    movel([0.121512, -1.277882, -2.639654, -0.794853, 1.570796, 1.692308],accel_mss,speed_ms,0,blend_radius_m)
    movel([0.121915, -1.277664, -2.639778, -0.794948, 1.570796, 1.692711],accel_mss,speed_ms,0,blend_radius_m)
    movel([0.122224, -1.277485, -2.639879, -0.795025, 1.570796, 1.693020],accel_mss,speed_ms,0,blend_radius_m)
    movel([0.122594, -1.277272, -2.639999, -0.795118, 1.570796, 1.693390],accel_mss,speed_ms,0,blend_radius_m)
    movel([0.122927, -1.277174, -2.640055, -0.795160, 1.570796, 1.693724],accel_mss,speed_ms,0,blend_radius_m)
    movel([0.123154, -1.277358, -2.639950, -0.795080, 1.570796, 1.693950],accel_mss,speed_ms,0,blend_radius_m)
    movel([0.122937, -1.277676, -2.639771, -0.794942, 1.570796, 1.693733],accel_mss,speed_ms,0,blend_radius_m)
    movel([0.122394, -1.277926, -2.639629, -0.794834, 1.570796, 1.693190],accel_mss,speed_ms,0,blend_radius_m)
    movel([0.122493, -1.278132, -2.639513, -0.794745, 1.570796, 1.693289],accel_mss,speed_ms,0,blend_radius_m)
    movel([0.122823, -1.278090, -2.639536, -0.794763, 1.570796, 1.693620],accel_mss,speed_ms,0,blend_radius_m)
    movel([0.123129, -1.277991, -2.639592, -0.794806, 1.570796, 1.693926],accel_mss,speed_ms,0,blend_radius_m)
    movel([0.123433, -1.277648, -2.639786, -0.794954, 1.570796, 1.694230],accel_mss,speed_ms,0,blend_radius_m)
    movel([0.123760, -1.277440, -2.639904, -0.795045, 1.570796, 1.694556],accel_mss,speed_ms,0,blend_radius_m)
    movel([0.124094, -1.277452, -2.639898, -0.795040, 1.570796, 1.694890],accel_mss,speed_ms,0,blend_radius_m)
    movel([0.124564, -1.277440, -2.639904, -0.795045, 1.570796, 1.695360],accel_mss,speed_ms,0,blend_radius_m)
    movel([0.125059, -1.277384, -2.639936, -0.795069, 1.570796, 1.695855],accel_mss,speed_ms,0,blend_radius_m)
    movel([0.125372, -1.277273, -2.639999, -0.795117, 1.570796, 1.696168],accel_mss,speed_ms,0,blend_radius_m)
    movel([0.125657, -1.277244, -2.640015, -0.795130, 1.570796, 1.696454],accel_mss,speed_ms,0,blend_radius_m)
    movel([0.125972, -1.277065, -2.640117, -0.795208, 1.570796, 1.696768],accel_mss,speed_ms,0,blend_radius_m)
    movel([0.126196, -1.277124, -2.640083, -0.795182, 1.570796, 1.696993],accel_mss,speed_ms,0,blend_radius_m)
    movel([0.126436, -1.277173, -2.640055, -0.795161, 1.570796, 1.697232],accel_mss,speed_ms,0,blend_radius_m)
    movel([0.126810, -1.277070, -2.640113, -0.795205, 1.570796, 1.697606],accel_mss,speed_ms,0,blend_radius_m)
    movel([0.127277, -1.276889, -2.640215, -0.795284, 1.570796, 1.698073],accel_mss,speed_ms,0,blend_radius_m)
    movel([0.127645, -1.276791, -2.640271, -0.795327, 1.570796, 1.698441],accel_mss,speed_ms,0,blend_radius_m)
    movel([0.128058, -1.276835, -2.640246, -0.795308, 1.570796, 1.698854],accel_mss,speed_ms,0,blend_radius_m)
    movel([0.128268, -1.276992, -2.640157, -0.795239, 1.570796, 1.699064],accel_mss,speed_ms,0,blend_radius_m)
    movel([0.128442, -1.277211, -2.640033, -0.795144, 1.570796, 1.699239],accel_mss,speed_ms,0,blend_radius_m)
    movel([0.128502, -1.277437, -2.639906, -0.795046, 1.570796, 1.699298],accel_mss,speed_ms,0,blend_radius_m)
    movel([0.128278, -1.277739, -2.639735, -0.794915, 1.570796, 1.699074],accel_mss,speed_ms,0,blend_radius_m)
    movel([0.128301, -1.278030, -2.639570, -0.794789, 1.570796, 1.699097],accel_mss,speed_ms,0,blend_radius_m)
    movel([0.128456, -1.278253, -2.639444, -0.794692, 1.570796, 1.699252],accel_mss,speed_ms,0,blend_radius_m)
    movel([0.128142, -1.278841, -2.639111, -0.794438, 1.570796, 1.698939],accel_mss,speed_ms,0,blend_radius_m)
    movel([0.127643, -1.279450, -2.638765, -0.794174, 1.570796, 1.698439],accel_mss,speed_ms,0,blend_radius_m)
    movel([0.127331, -1.279820, -2.638555, -0.794015, 1.570796, 1.698128],accel_mss,speed_ms,0,blend_radius_m)
    movel([0.127066, -1.280148, -2.638368, -0.793873, 1.570796, 1.697863],accel_mss,speed_ms,0,blend_radius_m)
    movel([0.126852, -1.280424, -2.638211, -0.793754, 1.570796, 1.697648],accel_mss,speed_ms,0,blend_radius_m)
    movel([0.126937, -1.280641, -2.638087, -0.793661, 1.570796, 1.697734],accel_mss,speed_ms,0,blend_radius_m)
    movel([0.127240, -1.280865, -2.637959, -0.793565, 1.570796, 1.698036],accel_mss,speed_ms,0,blend_radius_m)
    movel([0.127528, -1.281108, -2.637821, -0.793460, 1.570796, 1.698325],accel_mss,speed_ms,0,blend_radius_m)
    movel([0.127643, -1.281364, -2.637675, -0.793350, 1.570796, 1.698439],accel_mss,speed_ms,0,blend_radius_m)
    movel([0.127335, -1.281559, -2.637563, -0.793266, 1.570796, 1.698131],accel_mss,speed_ms,0,blend_radius_m)
    movel([0.127124, -1.281455, -2.637623, -0.793311, 1.570796, 1.697920],accel_mss,speed_ms,0,blend_radius_m)
    movel([0.126991, -1.281268, -2.637730, -0.793391, 1.570796, 1.697788],accel_mss,speed_ms,0,blend_radius_m)
    movel([0.126865, -1.281079, -2.637837, -0.793473, 1.570796, 1.697661],accel_mss,speed_ms,0,blend_radius_m)
    movel([0.126558, -1.281192, -2.637773, -0.793424, 1.570796, 1.697354],accel_mss,speed_ms,0,blend_radius_m)
    movel([0.126435, -1.280994, -2.637886, -0.793509, 1.570796, 1.697231],accel_mss,speed_ms,0,blend_radius_m)
    movel([0.126185, -1.280895, -2.637942, -0.793552, 1.570796, 1.696981],accel_mss,speed_ms,0,blend_radius_m)
    movel([0.126273, -1.280615, -2.638102, -0.793672, 1.570796, 1.697069],accel_mss,speed_ms,0,blend_radius_m)
    movel([0.126374, -1.280318, -2.638271, -0.793800, 1.570796, 1.697170],accel_mss,speed_ms,0,blend_radius_m)
    movel([0.126672, -1.280154, -2.638364, -0.793870, 1.570796, 1.697468],accel_mss,speed_ms,0,blend_radius_m)
    movel([0.126485, -1.280006, -2.638449, -0.793935, 1.570796, 1.697281],accel_mss,speed_ms,0,blend_radius_m)
    movel([0.126217, -1.280245, -2.638312, -0.793831, 1.570796, 1.697013],accel_mss,speed_ms,0,blend_radius_m)
    movel([0.125927, -1.280465, -2.638187, -0.793737, 1.570796, 1.696723],accel_mss,speed_ms,0,blend_radius_m)
    movel([0.125642, -1.280712, -2.638046, -0.793630, 1.570796, 1.696438],accel_mss,speed_ms,0,blend_radius_m)
    movel([0.125248, -1.280906, -2.637936, -0.793547, 1.570796, 1.696044],accel_mss,speed_ms,0,blend_radius_m)
    movel([0.124945, -1.281110, -2.637820, -0.793459, 1.570796, 1.695741],accel_mss,speed_ms,0,blend_radius_m)
    movel([0.124618, -1.281268, -2.637729, -0.793391, 1.570796, 1.695414],accel_mss,speed_ms,0,blend_radius_m)
    movel([0.124820, -1.281407, -2.637650, -0.793332, 1.570796, 1.695616],accel_mss,speed_ms,0,blend_radius_m)
    movel([0.125120, -1.281303, -2.637710, -0.793376, 1.570796, 1.695916],accel_mss,speed_ms,0,blend_radius_m)
    movel([0.125422, -1.281303, -2.637709, -0.793376, 1.570796, 1.696218],accel_mss,speed_ms,0,blend_radius_m)
    movel([0.125734, -1.281325, -2.637697, -0.793367, 1.570796, 1.696530],accel_mss,speed_ms,0,blend_radius_m)
    movel([0.125551, -1.281207, -2.637764, -0.793418, 1.570796, 1.696347],accel_mss,speed_ms,0,blend_radius_m)
    movel([0.125887, -1.281100, -2.637826, -0.793464, 1.570796, 1.696683],accel_mss,speed_ms,0,blend_radius_m)
    movel([0.126035, -1.281250, -2.637740, -0.793399, 1.570796, 1.696831],accel_mss,speed_ms,0,blend_radius_m)
    movel([0.126335, -1.281283, -2.637721, -0.793385, 1.570796, 1.697131],accel_mss,speed_ms,0,blend_radius_m)
    movel([0.126542, -1.281456, -2.637622, -0.793310, 1.570796, 1.697338],accel_mss,speed_ms,0,blend_radius_m)
    movel([0.126874, -1.281511, -2.637591, -0.793287, 1.570796, 1.697670],accel_mss,speed_ms,0,blend_radius_m)
    movel([0.127085, -1.281732, -2.637465, -0.793192, 1.570796, 1.697881],accel_mss,speed_ms,0,blend_radius_m)
    movel([0.126908, -1.282027, -2.637296, -0.793066, 1.570796, 1.697705],accel_mss,speed_ms,0,blend_radius_m)
    movel([0.126872, -1.282378, -2.637096, -0.792915, 1.570796, 1.697668],accel_mss,speed_ms,0,blend_radius_m)
    movel([0.126732, -1.282647, -2.636942, -0.792800, 1.570796, 1.697528],accel_mss,speed_ms,0,blend_radius_m)
    movel([0.127032, -1.282483, -2.637035, -0.792870, 1.570796, 1.697828],accel_mss,speed_ms,0,blend_radius_m)
    movel([0.127020, -1.282092, -2.637259, -0.793038, 1.570796, 1.697816],accel_mss,speed_ms,0,blend_radius_m)
    movel([0.127207, -1.281796, -2.637428, -0.793165, 1.570796, 1.698004],accel_mss,speed_ms,0,blend_radius_m)
    movel([0.127325, -1.281990, -2.637318, -0.793082, 1.570796, 1.698121],accel_mss,speed_ms,0,blend_radius_m)
    movel([0.127108, -1.282326, -2.637125, -0.792937, 1.570796, 1.697904],accel_mss,speed_ms,0,blend_radius_m)
    movel([0.127401, -1.282233, -2.637178, -0.792977, 1.570796, 1.698197],accel_mss,speed_ms,0,blend_radius_m)
    movel([0.127190, -1.282793, -2.636858, -0.792738, 1.570796, 1.697986],accel_mss,speed_ms,0,blend_radius_m)
    movel([0.126973, -1.283052, -2.636710, -0.792627, 1.570796, 1.697769],accel_mss,speed_ms,0,blend_radius_m)
    movel([0.126665, -1.283232, -2.636607, -0.792550, 1.570796, 1.697462],accel_mss,speed_ms,0,blend_radius_m)
    movel([0.126509, -1.283540, -2.636430, -0.792419, 1.570796, 1.697305],accel_mss,speed_ms,0,blend_radius_m)
    movel([0.126164, -1.283969, -2.636184, -0.792236, 1.570796, 1.696960],accel_mss,speed_ms,0,blend_radius_m)
    movel([0.125846, -1.284341, -2.635970, -0.792077, 1.570796, 1.696642],accel_mss,speed_ms,0,blend_radius_m)
    movel([0.126192, -1.284417, -2.635927, -0.792045, 1.570796, 1.696988],accel_mss,speed_ms,0,blend_radius_m)
    movel([0.126470, -1.284556, -2.635847, -0.791986, 1.570796, 1.697267],accel_mss,speed_ms,0,blend_radius_m)
    movel([0.126536, -1.284775, -2.635721, -0.791893, 1.570796, 1.697332],accel_mss,speed_ms,0,blend_radius_m)
    movel([0.126661, -1.284987, -2.635599, -0.791803, 1.570796, 1.697458],accel_mss,speed_ms,0,blend_radius_m)
    movel([0.126532, -1.285317, -2.635409, -0.791663, 1.570796, 1.697328],accel_mss,speed_ms,0,blend_radius_m)
    movel([0.126278, -1.285671, -2.635205, -0.791513, 1.570796, 1.697074],accel_mss,speed_ms,0,blend_radius_m)
    movel([0.125958, -1.286079, -2.634970, -0.791340, 1.570796, 1.696754],accel_mss,speed_ms,0,blend_radius_m)
    movel([0.125587, -1.286339, -2.634821, -0.791230, 1.570796, 1.696383],accel_mss,speed_ms,0,blend_radius_m)
    movel([0.125858, -1.286124, -2.634944, -0.791320, 1.570796, 1.696654],accel_mss,speed_ms,0,blend_radius_m)
    movel([0.125869, -1.285839, -2.635109, -0.791441, 1.570796, 1.696665],accel_mss,speed_ms,0,blend_radius_m)
    movel([0.126028, -1.285541, -2.635280, -0.791568, 1.570796, 1.696825],accel_mss,speed_ms,0,blend_radius_m)
    movel([0.126232, -1.285026, -2.635577, -0.791786, 1.570796, 1.697029],accel_mss,speed_ms,0,blend_radius_m)
    movel([0.126003, -1.284962, -2.635614, -0.791813, 1.570796, 1.696799],accel_mss,speed_ms,0,blend_radius_m)
    movel([0.125957, -1.284696, -2.635767, -0.791927, 1.570796, 1.696753],accel_mss,speed_ms,0,blend_radius_m)
    movel([0.125809, -1.284543, -2.635854, -0.791991, 1.570796, 1.696605],accel_mss,speed_ms,0,blend_radius_m)
    movel([0.125586, -1.284429, -2.635920, -0.792040, 1.570796, 1.696383],accel_mss,speed_ms,0,blend_radius_m)
    movel([0.125377, -1.284351, -2.635965, -0.792073, 1.570796, 1.696173],accel_mss,speed_ms,0,blend_radius_m)
    movel([0.125610, -1.284068, -2.636127, -0.792194, 1.570796, 1.696406],accel_mss,speed_ms,0,blend_radius_m)
    movel([0.125992, -1.283659, -2.636362, -0.792368, 1.570796, 1.696789],accel_mss,speed_ms,0,blend_radius_m)
    movel([0.126321, -1.283308, -2.636563, -0.792518, 1.570796, 1.697118],accel_mss,speed_ms,0,blend_radius_m)
    movel([0.126533, -1.282968, -2.636758, -0.792663, 1.570796, 1.697330],accel_mss,speed_ms,0,blend_radius_m)
    movel([0.126193, -1.283188, -2.636632, -0.792569, 1.570796, 1.696989],accel_mss,speed_ms,0,blend_radius_m)
    movel([0.125766, -1.283548, -2.636426, -0.792415, 1.570796, 1.696563],accel_mss,speed_ms,0,blend_radius_m)
    movel([0.125446, -1.283919, -2.636213, -0.792257, 1.570796, 1.696242],accel_mss,speed_ms,0,blend_radius_m)
    movel([0.125139, -1.284055, -2.636135, -0.792199, 1.570796, 1.695935],accel_mss,speed_ms,0,blend_radius_m)
    movel([0.124558, -1.284490, -2.635885, -0.792014, 1.570796, 1.695354],accel_mss,speed_ms,0,blend_radius_m)
    movel([0.124536, -1.284797, -2.635709, -0.791884, 1.570796, 1.695333],accel_mss,speed_ms,0,blend_radius_m)
    movel([0.124872, -1.284837, -2.635685, -0.791866, 1.570796, 1.695668],accel_mss,speed_ms,0,blend_radius_m)
    movel([0.125134, -1.284821, -2.635695, -0.791873, 1.570796, 1.695931],accel_mss,speed_ms,0,blend_radius_m)
    movel([0.125420, -1.284693, -2.635768, -0.791928, 1.570796, 1.696217],accel_mss,speed_ms,0,blend_radius_m)
    movel([0.125608, -1.284848, -2.635679, -0.791862, 1.570796, 1.696404],accel_mss,speed_ms,0,blend_radius_m)
    movel([0.125786, -1.285070, -2.635551, -0.791768, 1.570796, 1.696583],accel_mss,speed_ms,0,blend_radius_m)
    movel([0.125996, -1.285162, -2.635498, -0.791728, 1.570796, 1.696792],accel_mss,speed_ms,0,blend_radius_m)
    movel([0.125747, -1.285560, -2.635269, -0.791559, 1.570796, 1.696543],accel_mss,speed_ms,0,blend_radius_m)
    movel([0.125404, -1.285997, -2.635017, -0.791374, 1.570796, 1.696200],accel_mss,speed_ms,0,blend_radius_m)
    movel([0.125296, -1.286269, -2.634861, -0.791259, 1.570796, 1.696093],accel_mss,speed_ms,0,blend_radius_m)
    movel([0.124953, -1.286578, -2.634682, -0.791128, 1.570796, 1.695749],accel_mss,speed_ms,0,blend_radius_m)
    movel([0.124458, -1.286900, -2.634496, -0.790992, 1.570796, 1.695255],accel_mss,speed_ms,0,blend_radius_m)
    movel([0.123806, -1.287353, -2.634235, -0.790801, 1.570796, 1.694603],accel_mss,speed_ms,0,blend_radius_m)
    movel([0.124318, -1.287180, -2.634335, -0.790874, 1.570796, 1.695114],accel_mss,speed_ms,0,blend_radius_m)
    movel([0.124661, -1.287037, -2.634417, -0.790935, 1.570796, 1.695458],accel_mss,speed_ms,0,blend_radius_m)
    movel([0.124937, -1.286829, -2.634537, -0.791022, 1.570796, 1.695733],accel_mss,speed_ms,0,blend_radius_m)
    movel([0.125165, -1.286556, -2.634695, -0.791138, 1.570796, 1.695962],accel_mss,speed_ms,0,blend_radius_m)
    movel([0.125011, -1.286951, -2.634467, -0.790971, 1.570796, 1.695807],accel_mss,speed_ms,0,blend_radius_m)
    movel([0.124648, -1.287248, -2.634295, -0.790845, 1.570796, 1.695444],accel_mss,speed_ms,0,blend_radius_m)
    movel([0.124301, -1.287457, -2.634174, -0.790757, 1.570796, 1.695097],accel_mss,speed_ms,0,blend_radius_m)
    movel([0.123990, -1.287729, -2.634017, -0.790643, 1.570796, 1.694786],accel_mss,speed_ms,0,blend_radius_m)
    movel([0.123623, -1.287713, -2.634026, -0.790649, 1.570796, 1.694419],accel_mss,speed_ms,0,blend_radius_m)
    movel([0.123370, -1.287684, -2.634043, -0.790662, 1.570796, 1.694166],accel_mss,speed_ms,0,blend_radius_m)
    movel([0.122926, -1.288007, -2.633857, -0.790526, 1.570796, 1.693723],accel_mss,speed_ms,0,blend_radius_m)
    movel([0.122673, -1.288254, -2.633713, -0.790422, 1.570796, 1.693469],accel_mss,speed_ms,0,blend_radius_m)
    movel([0.122307, -1.288149, -2.633774, -0.790466, 1.570796, 1.693104],accel_mss,speed_ms,0,blend_radius_m)
    movel([0.122004, -1.288212, -2.633738, -0.790440, 1.570796, 1.692801],accel_mss,speed_ms,0,blend_radius_m)
    movel([0.121661, -1.288494, -2.633574, -0.790321, 1.570796, 1.692457],accel_mss,speed_ms,0,blend_radius_m)
    movel([0.121351, -1.288684, -2.633464, -0.790241, 1.570796, 1.692148],accel_mss,speed_ms,0,blend_radius_m)
    movel([0.121025, -1.288902, -2.633338, -0.790150, 1.570796, 1.691821],accel_mss,speed_ms,0,blend_radius_m)
    movel([0.120795, -1.289136, -2.633201, -0.790051, 1.570796, 1.691591],accel_mss,speed_ms,0,blend_radius_m)
    movel([0.120927, -1.288831, -2.633379, -0.790179, 1.570796, 1.691724],accel_mss,speed_ms,0,blend_radius_m)
    movel([0.120541, -1.288762, -2.633419, -0.790208, 1.570796, 1.691337],accel_mss,speed_ms,0,blend_radius_m)
    movel([0.120155, -1.288905, -2.633336, -0.790148, 1.570796, 1.690951],accel_mss,speed_ms,0,blend_radius_m)
    movel([0.119775, -1.289045, -2.633255, -0.790089, 1.570796, 1.690571],accel_mss,speed_ms,0,blend_radius_m)
    movel([0.119308, -1.289155, -2.633191, -0.790043, 1.570796, 1.690104],accel_mss,speed_ms,0,blend_radius_m)
    movel([0.119086, -1.289030, -2.633263, -0.790096, 1.570796, 1.689882],accel_mss,speed_ms,0,blend_radius_m)
    movel([0.118778, -1.288930, -2.633321, -0.790138, 1.570796, 1.689574],accel_mss,speed_ms,0,blend_radius_m)
    movel([0.118635, -1.288762, -2.633419, -0.790208, 1.570796, 1.689431],accel_mss,speed_ms,0,blend_radius_m)
    movel([0.118460, -1.288562, -2.633535, -0.790292, 1.570796, 1.689257],accel_mss,speed_ms,0,blend_radius_m)
    movel([0.118223, -1.288514, -2.633562, -0.790312, 1.570796, 1.689019],accel_mss,speed_ms,0,blend_radius_m)
    movel([0.118344, -1.288851, -2.633367, -0.790171, 1.570796, 1.689141],accel_mss,speed_ms,0,blend_radius_m)
    movel([0.118538, -1.289082, -2.633233, -0.790074, 1.570796, 1.689335],accel_mss,speed_ms,0,blend_radius_m)
    movel([0.118550, -1.289354, -2.633075, -0.789960, 1.570796, 1.689347],accel_mss,speed_ms,0,blend_radius_m)
    movel([0.118849, -1.289162, -2.633186, -0.790040, 1.570796, 1.689645],accel_mss,speed_ms,0,blend_radius_m)
    movel([0.118996, -1.289366, -2.633068, -0.789955, 1.570796, 1.689792],accel_mss,speed_ms,0,blend_radius_m)
    movel([0.118698, -1.289531, -2.632972, -0.789886, 1.570796, 1.689495],accel_mss,speed_ms,0,blend_radius_m)
    movel([0.118450, -1.289508, -2.632986, -0.789895, 1.570796, 1.689246],accel_mss,speed_ms,0,blend_radius_m)
    movel([0.118230, -1.289407, -2.633044, -0.789938, 1.570796, 1.689027],accel_mss,speed_ms,0,blend_radius_m)
    movel([0.118043, -1.289226, -2.633149, -0.790013, 1.570796, 1.688839],accel_mss,speed_ms,0,blend_radius_m)
    movel([0.117955, -1.289021, -2.633268, -0.790099, 1.570796, 1.688751],accel_mss,speed_ms,0,blend_radius_m)
    movel([0.118003, -1.288720, -2.633443, -0.790226, 1.570796, 1.688799],accel_mss,speed_ms,0,blend_radius_m)
    movel([0.118007, -1.288440, -2.633605, -0.790343, 1.570796, 1.688804],accel_mss,speed_ms,0,blend_radius_m)
    movel([0.118087, -1.288046, -2.633834, -0.790509, 1.570796, 1.688883],accel_mss,speed_ms,0,blend_radius_m)
    movel([0.118058, -1.287732, -2.634015, -0.790641, 1.570796, 1.688855],accel_mss,speed_ms,0,blend_radius_m)
    movel([0.117873, -1.287509, -2.634144, -0.790735, 1.570796, 1.688669],accel_mss,speed_ms,0,blend_radius_m)
    movel([0.117791, -1.287302, -2.634264, -0.790823, 1.570796, 1.688587],accel_mss,speed_ms,0,blend_radius_m)
    movel([0.117513, -1.287599, -2.634092, -0.790697, 1.570796, 1.688309],accel_mss,speed_ms,0,blend_radius_m)
    movel([0.117263, -1.287555, -2.634118, -0.790716, 1.570796, 1.688060],accel_mss,speed_ms,0,blend_radius_m)
    movel([0.116775, -1.287477, -2.634163, -0.790749, 1.570796, 1.687571],accel_mss,speed_ms,0,blend_radius_m)
    movel([0.116521, -1.287240, -2.634300, -0.790849, 1.570796, 1.687318],accel_mss,speed_ms,0,blend_radius_m)
    movel([0.116399, -1.286963, -2.634460, -0.790966, 1.570796, 1.687195],accel_mss,speed_ms,0,blend_radius_m)
    movel([0.116380, -1.286678, -2.634625, -0.791086, 1.570796, 1.687176],accel_mss,speed_ms,0,blend_radius_m)
    movel([0.116535, -1.286390, -2.634791, -0.791208, 1.570796, 1.687332],accel_mss,speed_ms,0,blend_radius_m)
    movel([0.116603, -1.286612, -2.634663, -0.791114, 1.570796, 1.687400],accel_mss,speed_ms,0,blend_radius_m)
    movel([0.116900, -1.286376, -2.634799, -0.791214, 1.570796, 1.687696],accel_mss,speed_ms,0,blend_radius_m)
    movel([0.116924, -1.286108, -2.634954, -0.791327, 1.570796, 1.687721],accel_mss,speed_ms,0,blend_radius_m)
    movel([0.116662, -1.286018, -2.635006, -0.791366, 1.570796, 1.687458],accel_mss,speed_ms,0,blend_radius_m)
    movel([0.117083, -1.285824, -2.635117, -0.791448, 1.570796, 1.687879],accel_mss,speed_ms,0,blend_radius_m)
    movel([0.117398, -1.285712, -2.635182, -0.791495, 1.570796, 1.688195],accel_mss,speed_ms,0,blend_radius_m)
    movel([0.117220, -1.285518, -2.635294, -0.791578, 1.570796, 1.688016],accel_mss,speed_ms,0,blend_radius_m)
    movel([0.116901, -1.285694, -2.635192, -0.791503, 1.570796, 1.687697],accel_mss,speed_ms,0,blend_radius_m)
    movel([0.117066, -1.285357, -2.635386, -0.791646, 1.570796, 1.687862],accel_mss,speed_ms,0,blend_radius_m)
    movel([0.117091, -1.285021, -2.635580, -0.791789, 1.570796, 1.687888],accel_mss,speed_ms,0,blend_radius_m)
    movel([0.117345, -1.284667, -2.635783, -0.791939, 1.570796, 1.688141],accel_mss,speed_ms,0,blend_radius_m)
    movel([0.117730, -1.284770, -2.635724, -0.791895, 1.570796, 1.688526],accel_mss,speed_ms,0,blend_radius_m)
    movel([0.117907, -1.284892, -2.635654, -0.791843, 1.570796, 1.688704],accel_mss,speed_ms,0,blend_radius_m)
    movel([0.118256, -1.284658, -2.635788, -0.791942, 1.570796, 1.689052],accel_mss,speed_ms,0,blend_radius_m)
    movel([0.118549, -1.284539, -2.635857, -0.791993, 1.570796, 1.689345],accel_mss,speed_ms,0,blend_radius_m)
    movel([0.118546, -1.284272, -2.636010, -0.792107, 1.570796, 1.689343],accel_mss,speed_ms,0,blend_radius_m)
    movel([0.118238, -1.284183, -2.636061, -0.792145, 1.570796, 1.689034],accel_mss,speed_ms,0,blend_radius_m)
    movel([0.117886, -1.284442, -2.635912, -0.792034, 1.570796, 1.688682],accel_mss,speed_ms,0,blend_radius_m)
    movel([0.117733, -1.284271, -2.636011, -0.792107, 1.570796, 1.688530],accel_mss,speed_ms,0,blend_radius_m)
    movel([0.117417, -1.284364, -2.635957, -0.792068, 1.570796, 1.688213],accel_mss,speed_ms,0,blend_radius_m)
    movel([0.117154, -1.284337, -2.635973, -0.792079, 1.570796, 1.687950],accel_mss,speed_ms,0,blend_radius_m)
    movel([0.117279, -1.284512, -2.635872, -0.792005, 1.570796, 1.688075],accel_mss,speed_ms,0,blend_radius_m)
    movel([0.117007, -1.284738, -2.635742, -0.791908, 1.570796, 1.687803],accel_mss,speed_ms,0,blend_radius_m)
    movel([0.116841, -1.284482, -2.635890, -0.792018, 1.570796, 1.687638],accel_mss,speed_ms,0,blend_radius_m)
    movel([0.116572, -1.284442, -2.635912, -0.792034, 1.570796, 1.687368],accel_mss,speed_ms,0,blend_radius_m)
    movel([0.116208, -1.284321, -2.635982, -0.792086, 1.570796, 1.687004],accel_mss,speed_ms,0,blend_radius_m)
    movel([0.116016, -1.284221, -2.636040, -0.792129, 1.570796, 1.686813],accel_mss,speed_ms,0,blend_radius_m)
    movel([0.115720, -1.284016, -2.636157, -0.792216, 1.570796, 1.686516],accel_mss,speed_ms,0,blend_radius_m)
    movel([0.115647, -1.283805, -2.636278, -0.792306, 1.570796, 1.686444],accel_mss,speed_ms,0,blend_radius_m)
    movel([0.115443, -1.283672, -2.636355, -0.792363, 1.570796, 1.686240],accel_mss,speed_ms,0,blend_radius_m)
    movel([0.115403, -1.283946, -2.636197, -0.792246, 1.570796, 1.686199],accel_mss,speed_ms,0,blend_radius_m)
    movel([0.115514, -1.284149, -2.636081, -0.792159, 1.570796, 1.686310],accel_mss,speed_ms,0,blend_radius_m)
    movel([0.115629, -1.284337, -2.635973, -0.792079, 1.570796, 1.686426],accel_mss,speed_ms,0,blend_radius_m)
    movel([0.115390, -1.284585, -2.635830, -0.791974, 1.570796, 1.686186],accel_mss,speed_ms,0,blend_radius_m)
    movel([0.115503, -1.284298, -2.635995, -0.792096, 1.570796, 1.686299],accel_mss,speed_ms,0,blend_radius_m)
    movel([0.115218, -1.284249, -2.636023, -0.792117, 1.570796, 1.686014],accel_mss,speed_ms,0,blend_radius_m)
    movel([0.115021, -1.284085, -2.636118, -0.792187, 1.570796, 1.685817],accel_mss,speed_ms,0,blend_radius_m)
    movel([0.115096, -1.283727, -2.636323, -0.792339, 1.570796, 1.685893],accel_mss,speed_ms,0,blend_radius_m)
    movel([0.115346, -1.283483, -2.636463, -0.792443, 1.570796, 1.686143],accel_mss,speed_ms,0,blend_radius_m)
    movel([0.115659, -1.283298, -2.636569, -0.792522, 1.570796, 1.686455],accel_mss,speed_ms,0,blend_radius_m)
    movel([0.115744, -1.283014, -2.636731, -0.792643, 1.570796, 1.686541],accel_mss,speed_ms,0,blend_radius_m)
    movel([0.115466, -1.283019, -2.636729, -0.792641, 1.570796, 1.686262],accel_mss,speed_ms,0,blend_radius_m)
    movel([0.115654, -1.283150, -2.636654, -0.792585, 1.570796, 1.686450],accel_mss,speed_ms,0,blend_radius_m)
    movel([0.115361, -1.283311, -2.636561, -0.792516, 1.570796, 1.686157],accel_mss,speed_ms,0,blend_radius_m)
    movel([0.115061, -1.283543, -2.636429, -0.792418, 1.570796, 1.685857],accel_mss,speed_ms,0,blend_radius_m)
    movel([0.115080, -1.283227, -2.636610, -0.792552, 1.570796, 1.685876],accel_mss,speed_ms,0,blend_radius_m)
    movel([0.115258, -1.282848, -2.636827, -0.792714, 1.570796, 1.686055],accel_mss,speed_ms,0,blend_radius_m)
    movel([0.115654, -1.282292, -2.637144, -0.792952, 1.570796, 1.686451],accel_mss,speed_ms,0,blend_radius_m)
    movel([0.116074, -1.281785, -2.637435, -0.793170, 1.570796, 1.686870],accel_mss,speed_ms,0,blend_radius_m)
    movel([0.116426, -1.281592, -2.637545, -0.793252, 1.570796, 1.687222],accel_mss,speed_ms,0,blend_radius_m)
    movel([0.116646, -1.281315, -2.637702, -0.793371, 1.570796, 1.687442],accel_mss,speed_ms,0,blend_radius_m)
    movel([0.116582, -1.281620, -2.637529, -0.793240, 1.570796, 1.687378],accel_mss,speed_ms,0,blend_radius_m)
    movel([0.116643, -1.281835, -2.637406, -0.793148, 1.570796, 1.687439],accel_mss,speed_ms,0,blend_radius_m)
    movel([0.116707, -1.281553, -2.637567, -0.793269, 1.570796, 1.687503],accel_mss,speed_ms,0,blend_radius_m)
    movel([0.116909, -1.281226, -2.637753, -0.793409, 1.570796, 1.687705],accel_mss,speed_ms,0,blend_radius_m)
    movel([0.117205, -1.280821, -2.637985, -0.793584, 1.570796, 1.688001],accel_mss,speed_ms,0,blend_radius_m)
    movel([0.117543, -1.280489, -2.638173, -0.793726, 1.570796, 1.688340],accel_mss,speed_ms,0,blend_radius_m)
    movel([0.117995, -1.280116, -2.638386, -0.793887, 1.570796, 1.688792],accel_mss,speed_ms,0,blend_radius_m)
    movel([0.118505, -1.279759, -2.638589, -0.794041, 1.570796, 1.689301],accel_mss,speed_ms,0,blend_radius_m)
    movel([0.118905, -1.279558, -2.638703, -0.794128, 1.570796, 1.689701],accel_mss,speed_ms,0,blend_radius_m)
    movel([0.119186, -1.279400, -2.638793, -0.794196, 1.570796, 1.689982],accel_mss,speed_ms,0,blend_radius_m)
    movel([0.119588, -1.278941, -2.639054, -0.794394, 1.570796, 1.690384],accel_mss,speed_ms,0,blend_radius_m)
    movel([0.120097, -1.278618, -2.639237, -0.794534, 1.570796, 1.690893],accel_mss,speed_ms,0,blend_radius_m)
    movel([0.120709, -1.278294, -2.639421, -0.794674, 1.570796, 1.691505],accel_mss,speed_ms,0,blend_radius_m)
    speed_ms = 0.003
    movel([0.120709, -1.264276, -2.632718, -0.815395, 1.570796, 1.691505],accel_mss,speed_ms,0,blend_radius_m)
    speed_ms = 1.000
    movel([0.120709, -1.237636, -2.618929, -0.855824, 1.570796, 1.691505],accel_mss,speed_ms,0,blend_radius_m)
    movel([0.125841, -1.252553, -2.610810, -0.849026, 1.570796, 1.696637],accel_mss,speed_ms,0,blend_radius_m)
    movel([0.125841, -1.279005, -2.624402, -0.808983, 1.570796, 1.696637],accel_mss,speed_ms,0,blend_radius_m)
    speed_ms = 0.003
    movel([0.125841, -1.289387, -2.629367, -0.793635, 1.570796, 1.696637],accel_mss,speed_ms,0,blend_radius_m)
    speed_ms = 0.007
    movel([0.126409, -1.289203, -2.629473, -0.793712, 1.570796, 1.697205],accel_mss,speed_ms,0,blend_radius_m)
    movel([0.126885, -1.289319, -2.629406, -0.793664, 1.570796, 1.697681],accel_mss,speed_ms,0,blend_radius_m)
    movel([0.127106, -1.289596, -2.629245, -0.793548, 1.570796, 1.697902],accel_mss,speed_ms,0,blend_radius_m)
    movel([0.127129, -1.289972, -2.629026, -0.793391, 1.570796, 1.697926],accel_mss,speed_ms,0,blend_radius_m)
    movel([0.126949, -1.290402, -2.628775, -0.793212, 1.570796, 1.697745],accel_mss,speed_ms,0,blend_radius_m)
    movel([0.126587, -1.290840, -2.628519, -0.793030, 1.570796, 1.697383],accel_mss,speed_ms,0,blend_radius_m)
    movel([0.126157, -1.291198, -2.628310, -0.792881, 1.570796, 1.696953],accel_mss,speed_ms,0,blend_radius_m)
    movel([0.125815, -1.291362, -2.628214, -0.792813, 1.570796, 1.696612],accel_mss,speed_ms,0,blend_radius_m)
    movel([0.125497, -1.291358, -2.628216, -0.792814, 1.570796, 1.696294],accel_mss,speed_ms,0,blend_radius_m)
    movel([0.125147, -1.291186, -2.628317, -0.792886, 1.570796, 1.695944],accel_mss,speed_ms,0,blend_radius_m)
    movel([0.124917, -1.291011, -2.628419, -0.792959, 1.570796, 1.695713],accel_mss,speed_ms,0,blend_radius_m)
    movel([0.124836, -1.290718, -2.628590, -0.793081, 1.570796, 1.695632],accel_mss,speed_ms,0,blend_radius_m)
    movel([0.124930, -1.290446, -2.628749, -0.793194, 1.570796, 1.695726],accel_mss,speed_ms,0,blend_radius_m)
    movel([0.125307, -1.289838, -2.629104, -0.793447, 1.570796, 1.696103],accel_mss,speed_ms,0,blend_radius_m)
    movel([0.125841, -1.289387, -2.629367, -0.793635, 1.570796, 1.696637],accel_mss,speed_ms,0,blend_radius_m)
    speed_ms = 0.003
    movel([0.125841, -1.292905, -2.631005, -0.788479, 1.570796, 1.696637],accel_mss,speed_ms,0,blend_radius_m)
    speed_ms = 0.007
    movel([0.126409, -1.292722, -2.631112, -0.788555, 1.570796, 1.697205],accel_mss,speed_ms,0,blend_radius_m)
    movel([0.126885, -1.292837, -2.631045, -0.788507, 1.570796, 1.697681],accel_mss,speed_ms,0,blend_radius_m)
    movel([0.127106, -1.293114, -2.630883, -0.788393, 1.570796, 1.697902],accel_mss,speed_ms,0,blend_radius_m)
    movel([0.127129, -1.293488, -2.630663, -0.788237, 1.570796, 1.697926],accel_mss,speed_ms,0,blend_radius_m)
    movel([0.126949, -1.293918, -2.630411, -0.788060, 1.570796, 1.697745],accel_mss,speed_ms,0,blend_radius_m)
    movel([0.126587, -1.294354, -2.630155, -0.787879, 1.570796, 1.697383],accel_mss,speed_ms,0,blend_radius_m)
    movel([0.126157, -1.294712, -2.629945, -0.787732, 1.570796, 1.696953],accel_mss,speed_ms,0,blend_radius_m)
    movel([0.125815, -1.294875, -2.629849, -0.787665, 1.570796, 1.696612],accel_mss,speed_ms,0,blend_radius_m)
    movel([0.125497, -1.294872, -2.629851, -0.787666, 1.570796, 1.696294],accel_mss,speed_ms,0,blend_radius_m)
    movel([0.125147, -1.294700, -2.629952, -0.787737, 1.570796, 1.695944],accel_mss,speed_ms,0,blend_radius_m)
    movel([0.124917, -1.294525, -2.630055, -0.787809, 1.570796, 1.695713],accel_mss,speed_ms,0,blend_radius_m)
    movel([0.124836, -1.294233, -2.630226, -0.787930, 1.570796, 1.695632],accel_mss,speed_ms,0,blend_radius_m)
    movel([0.124930, -1.293961, -2.630386, -0.788042, 1.570796, 1.695726],accel_mss,speed_ms,0,blend_radius_m)
    movel([0.125307, -1.293354, -2.630742, -0.788293, 1.570796, 1.696103],accel_mss,speed_ms,0,blend_radius_m)
    movel([0.125841, -1.292905, -2.631005, -0.788479, 1.570796, 1.696637],accel_mss,speed_ms,0,blend_radius_m)
    speed_ms = 0.003
    movel([0.125841, -1.279005, -2.624402, -0.808983, 1.570796, 1.696637],accel_mss,speed_ms,0,blend_radius_m)
    speed_ms = 1.000
    movel([0.125841, -1.252553, -2.610810, -0.849026, 1.570796, 1.696637],accel_mss,speed_ms,0,blend_radius_m)
    movel([0.125714, -1.252259, -2.610972, -0.849158, 1.570796, 1.696510],accel_mss,speed_ms,0,blend_radius_m)
    movel([0.125714, -1.278714, -2.624568, -0.809107, 1.570796, 1.696510],accel_mss,speed_ms,0,blend_radius_m)
    speed_ms = 0.003
    movel([0.125714, -1.289098, -2.629535, -0.793756, 1.570796, 1.696510],accel_mss,speed_ms,0,blend_radius_m)
    speed_ms = 0.007
    movel([0.125116, -1.289566, -2.629262, -0.793561, 1.570796, 1.695913],accel_mss,speed_ms,0,blend_radius_m)
    movel([0.124690, -1.289934, -2.629048, -0.793407, 1.570796, 1.695486],accel_mss,speed_ms,0,blend_radius_m)
    movel([0.124387, -1.290122, -2.628938, -0.793329, 1.570796, 1.695184],accel_mss,speed_ms,0,blend_radius_m)
    movel([0.124112, -1.290192, -2.628897, -0.793299, 1.570796, 1.694908],accel_mss,speed_ms,0,blend_radius_m)
    movel([0.123791, -1.290167, -2.628912, -0.793310, 1.570796, 1.694587],accel_mss,speed_ms,0,blend_radius_m)
    movel([0.123486, -1.290105, -2.628948, -0.793336, 1.570796, 1.694282],accel_mss,speed_ms,0,blend_radius_m)
    movel([0.123975, -1.289797, -2.629128, -0.793464, 1.570796, 1.694771],accel_mss,speed_ms,0,blend_radius_m)
    movel([0.124421, -1.289476, -2.629315, -0.793598, 1.570796, 1.695218],accel_mss,speed_ms,0,blend_radius_m)
    movel([0.124814, -1.289137, -2.629512, -0.793740, 1.570796, 1.695611],accel_mss,speed_ms,0,blend_radius_m)
    movel([0.125102, -1.288757, -2.629733, -0.793899, 1.570796, 1.695898],accel_mss,speed_ms,0,blend_radius_m)
    movel([0.125154, -1.288288, -2.630006, -0.794095, 1.570796, 1.695950],accel_mss,speed_ms,0,blend_radius_m)
    movel([0.125185, -1.287892, -2.630236, -0.794261, 1.570796, 1.695982],accel_mss,speed_ms,0,blend_radius_m)
    movel([0.125395, -1.287628, -2.630389, -0.794372, 1.570796, 1.696192],accel_mss,speed_ms,0,blend_radius_m)
    movel([0.125877, -1.287749, -2.630319, -0.794321, 1.570796, 1.696673],accel_mss,speed_ms,0,blend_radius_m)
    movel([0.126153, -1.287866, -2.630251, -0.794272, 1.570796, 1.696950],accel_mss,speed_ms,0,blend_radius_m)
    movel([0.126429, -1.287990, -2.630179, -0.794220, 1.570796, 1.697225],accel_mss,speed_ms,0,blend_radius_m)
    movel([0.126681, -1.288087, -2.630122, -0.794179, 1.570796, 1.697477],accel_mss,speed_ms,0,blend_radius_m)
    movel([0.126897, -1.288163, -2.630078, -0.794148, 1.570796, 1.697693],accel_mss,speed_ms,0,blend_radius_m)
    movel([0.127229, -1.287958, -2.630197, -0.794234, 1.570796, 1.698026],accel_mss,speed_ms,0,blend_radius_m)
    movel([0.127674, -1.287524, -2.630449, -0.794416, 1.570796, 1.698471],accel_mss,speed_ms,0,blend_radius_m)
    movel([0.128128, -1.287086, -2.630703, -0.794600, 1.570796, 1.698925],accel_mss,speed_ms,0,blend_radius_m)
    movel([0.128429, -1.286881, -2.630822, -0.794686, 1.570796, 1.699226],accel_mss,speed_ms,0,blend_radius_m)
    movel([0.128504, -1.287122, -2.630682, -0.794585, 1.570796, 1.699300],accel_mss,speed_ms,0,blend_radius_m)
    movel([0.128372, -1.287487, -2.630471, -0.794431, 1.570796, 1.699168],accel_mss,speed_ms,0,blend_radius_m)
    movel([0.128339, -1.287789, -2.630295, -0.794304, 1.570796, 1.699136],accel_mss,speed_ms,0,blend_radius_m)
    movel([0.128414, -1.288014, -2.630165, -0.794210, 1.570796, 1.699210],accel_mss,speed_ms,0,blend_radius_m)
    movel([0.128583, -1.288152, -2.630085, -0.794152, 1.570796, 1.699379],accel_mss,speed_ms,0,blend_radius_m)
    movel([0.128788, -1.288331, -2.629981, -0.794077, 1.570796, 1.699585],accel_mss,speed_ms,0,blend_radius_m)
    movel([0.128564, -1.288855, -2.629676, -0.793858, 1.570796, 1.699361],accel_mss,speed_ms,0,blend_radius_m)
    movel([0.128374, -1.289234, -2.629456, -0.793699, 1.570796, 1.699171],accel_mss,speed_ms,0,blend_radius_m)
    movel([0.128578, -1.289538, -2.629279, -0.793572, 1.570796, 1.699374],accel_mss,speed_ms,0,blend_radius_m)
    movel([0.128904, -1.289561, -2.629265, -0.793563, 1.570796, 1.699700],accel_mss,speed_ms,0,blend_radius_m)
    movel([0.129249, -1.289473, -2.629316, -0.793599, 1.570796, 1.700045],accel_mss,speed_ms,0,blend_radius_m)
    movel([0.129556, -1.289459, -2.629324, -0.793605, 1.570796, 1.700352],accel_mss,speed_ms,0,blend_radius_m)
    movel([0.128946, -1.290192, -2.628897, -0.793300, 1.570796, 1.699742],accel_mss,speed_ms,0,blend_radius_m)
    movel([0.128535, -1.290671, -2.628618, -0.793100, 1.570796, 1.699331],accel_mss,speed_ms,0,blend_radius_m)
    movel([0.128325, -1.291040, -2.628402, -0.792947, 1.570796, 1.699122],accel_mss,speed_ms,0,blend_radius_m)
    movel([0.128288, -1.291354, -2.628218, -0.792816, 1.570796, 1.699085],accel_mss,speed_ms,0,blend_radius_m)
    movel([0.128402, -1.291671, -2.628033, -0.792685, 1.570796, 1.699198],accel_mss,speed_ms,0,blend_radius_m)
    movel([0.128567, -1.291995, -2.627843, -0.792550, 1.570796, 1.699364],accel_mss,speed_ms,0,blend_radius_m)
    movel([0.127935, -1.291898, -2.627900, -0.792591, 1.570796, 1.698731],accel_mss,speed_ms,0,blend_radius_m)
    movel([0.127455, -1.291638, -2.628052, -0.792698, 1.570796, 1.698251],accel_mss,speed_ms,0,blend_radius_m)
    movel([0.127078, -1.291605, -2.628072, -0.792712, 1.570796, 1.697874],accel_mss,speed_ms,0,blend_radius_m)
    movel([0.126768, -1.291773, -2.627974, -0.792642, 1.570796, 1.697564],accel_mss,speed_ms,0,blend_radius_m)
    movel([0.126509, -1.292126, -2.627767, -0.792496, 1.570796, 1.697305],accel_mss,speed_ms,0,blend_radius_m)
    movel([0.126305, -1.292441, -2.627582, -0.792366, 1.570796, 1.697101],accel_mss,speed_ms,0,blend_radius_m)
    movel([0.126018, -1.292652, -2.627459, -0.792279, 1.570796, 1.696815],accel_mss,speed_ms,0,blend_radius_m)
    movel([0.125705, -1.292923, -2.627299, -0.792166, 1.570796, 1.696501],accel_mss,speed_ms,0,blend_radius_m)
    movel([0.125159, -1.293525, -2.626946, -0.791918, 1.570796, 1.695956],accel_mss,speed_ms,0,blend_radius_m)
    movel([0.125190, -1.293230, -2.627119, -0.792040, 1.570796, 1.695986],accel_mss,speed_ms,0,blend_radius_m)
    movel([0.125220, -1.292676, -2.627445, -0.792269, 1.570796, 1.696016],accel_mss,speed_ms,0,blend_radius_m)
    movel([0.125143, -1.292389, -2.627612, -0.792387, 1.570796, 1.695940],accel_mss,speed_ms,0,blend_radius_m)
    movel([0.124950, -1.292291, -2.627670, -0.792428, 1.570796, 1.695747],accel_mss,speed_ms,0,blend_radius_m)
    movel([0.124630, -1.292344, -2.627639, -0.792406, 1.570796, 1.695427],accel_mss,speed_ms,0,blend_radius_m)
    movel([0.124057, -1.292535, -2.627527, -0.792327, 1.570796, 1.694854],accel_mss,speed_ms,0,blend_radius_m)
    movel([0.123746, -1.292485, -2.627556, -0.792347, 1.570796, 1.694542],accel_mss,speed_ms,0,blend_radius_m)
    movel([0.123747, -1.292097, -2.627784, -0.792508, 1.570796, 1.694543],accel_mss,speed_ms,0,blend_radius_m)
    movel([0.123613, -1.291854, -2.627926, -0.792609, 1.570796, 1.694410],accel_mss,speed_ms,0,blend_radius_m)
    movel([0.123150, -1.291655, -2.628042, -0.792691, 1.570796, 1.693946],accel_mss,speed_ms,0,blend_radius_m)
    movel([0.123672, -1.291292, -2.628255, -0.792842, 1.570796, 1.694469],accel_mss,speed_ms,0,blend_radius_m)
    movel([0.124196, -1.290929, -2.628467, -0.792993, 1.570796, 1.694992],accel_mss,speed_ms,0,blend_radius_m)
    movel([0.124474, -1.291314, -2.628242, -0.792833, 1.570796, 1.695270],accel_mss,speed_ms,0,blend_radius_m)
    movel([0.124862, -1.291670, -2.628034, -0.792685, 1.570796, 1.695659],accel_mss,speed_ms,0,blend_radius_m)
    movel([0.125351, -1.291794, -2.627961, -0.792634, 1.570796, 1.696148],accel_mss,speed_ms,0,blend_radius_m)
    movel([0.125916, -1.291682, -2.628027, -0.792680, 1.570796, 1.696713],accel_mss,speed_ms,0,blend_radius_m)
    movel([0.126523, -1.291346, -2.628223, -0.792819, 1.570796, 1.697320],accel_mss,speed_ms,0,blend_radius_m)
    movel([0.126930, -1.291005, -2.628423, -0.792961, 1.570796, 1.697726],accel_mss,speed_ms,0,blend_radius_m)
    movel([0.127231, -1.290641, -2.628635, -0.793112, 1.570796, 1.698027],accel_mss,speed_ms,0,blend_radius_m)
    movel([0.127430, -1.290246, -2.628866, -0.793277, 1.570796, 1.698227],accel_mss,speed_ms,0,blend_radius_m)
    movel([0.127541, -1.289803, -2.629124, -0.793462, 1.570796, 1.698338],accel_mss,speed_ms,0,blend_radius_m)
    movel([0.127562, -1.289505, -2.629298, -0.793586, 1.570796, 1.698359],accel_mss,speed_ms,0,blend_radius_m)
    movel([0.127420, -1.289144, -2.629508, -0.793737, 1.570796, 1.698216],accel_mss,speed_ms,0,blend_radius_m)
    movel([0.127207, -1.288974, -2.629607, -0.793808, 1.570796, 1.698004],accel_mss,speed_ms,0,blend_radius_m)
    movel([0.126764, -1.288800, -2.629708, -0.793881, 1.570796, 1.697560],accel_mss,speed_ms,0,blend_radius_m)
    movel([0.126263, -1.288841, -2.629684, -0.793864, 1.570796, 1.697060],accel_mss,speed_ms,0,blend_radius_m)
    movel([0.125714, -1.289098, -2.629535, -0.793756, 1.570796, 1.696510],accel_mss,speed_ms,0,blend_radius_m)
    speed_ms = 0.003
    movel([0.125714, -1.292616, -2.631174, -0.788599, 1.570796, 1.696510],accel_mss,speed_ms,0,blend_radius_m)
    speed_ms = 0.007
    movel([0.125116, -1.293083, -2.630900, -0.788405, 1.570796, 1.695913],accel_mss,speed_ms,0,blend_radius_m)
    movel([0.124690, -1.293450, -2.630686, -0.788253, 1.570796, 1.695486],accel_mss,speed_ms,0,blend_radius_m)
    movel([0.124387, -1.293638, -2.630575, -0.788175, 1.570796, 1.695184],accel_mss,speed_ms,0,blend_radius_m)
    movel([0.124112, -1.293708, -2.630534, -0.788146, 1.570796, 1.694908],accel_mss,speed_ms,0,blend_radius_m)
    movel([0.123791, -1.293683, -2.630549, -0.788157, 1.570796, 1.694587],accel_mss,speed_ms,0,blend_radius_m)
    movel([0.123486, -1.293622, -2.630585, -0.788182, 1.570796, 1.694282],accel_mss,speed_ms,0,blend_radius_m)
    movel([0.123975, -1.293314, -2.630765, -0.788310, 1.570796, 1.694771],accel_mss,speed_ms,0,blend_radius_m)
    movel([0.124421, -1.292993, -2.630953, -0.788443, 1.570796, 1.695218],accel_mss,speed_ms,0,blend_radius_m)
    movel([0.124814, -1.292655, -2.631151, -0.788583, 1.570796, 1.695611],accel_mss,speed_ms,0,blend_radius_m)
    movel([0.125102, -1.292276, -2.631373, -0.788740, 1.570796, 1.695898],accel_mss,speed_ms,0,blend_radius_m)
    movel([0.125154, -1.291808, -2.631646, -0.788935, 1.570796, 1.695950],accel_mss,speed_ms,0,blend_radius_m)
    movel([0.125185, -1.291413, -2.631877, -0.789099, 1.570796, 1.695982],accel_mss,speed_ms,0,blend_radius_m)
    movel([0.125395, -1.291150, -2.632030, -0.789209, 1.570796, 1.696192],accel_mss,speed_ms,0,blend_radius_m)
    movel([0.125877, -1.291270, -2.631960, -0.789159, 1.570796, 1.696673],accel_mss,speed_ms,0,blend_radius_m)
    movel([0.126153, -1.291387, -2.631892, -0.789110, 1.570796, 1.696950],accel_mss,speed_ms,0,blend_radius_m)
    movel([0.126429, -1.291511, -2.631820, -0.789059, 1.570796, 1.697225],accel_mss,speed_ms,0,blend_radius_m)
    movel([0.126681, -1.291608, -2.631763, -0.789018, 1.570796, 1.697477],accel_mss,speed_ms,0,blend_radius_m)
    movel([0.126897, -1.291683, -2.631719, -0.788987, 1.570796, 1.697693],accel_mss,speed_ms,0,blend_radius_m)
    movel([0.127229, -1.291479, -2.631838, -0.789072, 1.570796, 1.698026],accel_mss,speed_ms,0,blend_radius_m)
    movel([0.127674, -1.291046, -2.632091, -0.789252, 1.570796, 1.698471],accel_mss,speed_ms,0,blend_radius_m)
    movel([0.128128, -1.290608, -2.632346, -0.789435, 1.570796, 1.698925],accel_mss,speed_ms,0,blend_radius_m)
    movel([0.128429, -1.290404, -2.632465, -0.789520, 1.570796, 1.699226],accel_mss,speed_ms,0,blend_radius_m)
    movel([0.128504, -1.290645, -2.632325, -0.789420, 1.570796, 1.699300],accel_mss,speed_ms,0,blend_radius_m)
    movel([0.128372, -1.291008, -2.632113, -0.789268, 1.570796, 1.699168],accel_mss,speed_ms,0,blend_radius_m)
    movel([0.128339, -1.291311, -2.631936, -0.789142, 1.570796, 1.699136],accel_mss,speed_ms,0,blend_radius_m)
    movel([0.128414, -1.291535, -2.631806, -0.789049, 1.570796, 1.699210],accel_mss,speed_ms,0,blend_radius_m)
    movel([0.128583, -1.291672, -2.631725, -0.788991, 1.570796, 1.699379],accel_mss,speed_ms,0,blend_radius_m)
    movel([0.128788, -1.291851, -2.631621, -0.788917, 1.570796, 1.699585],accel_mss,speed_ms,0,blend_radius_m)
    movel([0.128564, -1.292374, -2.631316, -0.788700, 1.570796, 1.699361],accel_mss,speed_ms,0,blend_radius_m)
    movel([0.128374, -1.292752, -2.631095, -0.788543, 1.570796, 1.699171],accel_mss,speed_ms,0,blend_radius_m)
    movel([0.128578, -1.293056, -2.630917, -0.788417, 1.570796, 1.699374],accel_mss,speed_ms,0,blend_radius_m)
    movel([0.128904, -1.293079, -2.630903, -0.788407, 1.570796, 1.699700],accel_mss,speed_ms,0,blend_radius_m)
    movel([0.129249, -1.292991, -2.630955, -0.788443, 1.570796, 1.700045],accel_mss,speed_ms,0,blend_radius_m)
    movel([0.129556, -1.292977, -2.630963, -0.788449, 1.570796, 1.700352],accel_mss,speed_ms,0,blend_radius_m)
    movel([0.128946, -1.293708, -2.630534, -0.788147, 1.570796, 1.699742],accel_mss,speed_ms,0,blend_radius_m)
    movel([0.128535, -1.294185, -2.630254, -0.787949, 1.570796, 1.699331],accel_mss,speed_ms,0,blend_radius_m)
    movel([0.128325, -1.294554, -2.630038, -0.787797, 1.570796, 1.699122],accel_mss,speed_ms,0,blend_radius_m)
    movel([0.128288, -1.294868, -2.629854, -0.787668, 1.570796, 1.699085],accel_mss,speed_ms,0,blend_radius_m)
    movel([0.128402, -1.295183, -2.629668, -0.787538, 1.570796, 1.699198],accel_mss,speed_ms,0,blend_radius_m)
    movel([0.128567, -1.295507, -2.629477, -0.787404, 1.570796, 1.699364],accel_mss,speed_ms,0,blend_radius_m)
    movel([0.127935, -1.295410, -2.629534, -0.787444, 1.570796, 1.698731],accel_mss,speed_ms,0,blend_radius_m)
    movel([0.127455, -1.295151, -2.629687, -0.787551, 1.570796, 1.698251],accel_mss,speed_ms,0,blend_radius_m)
    movel([0.127078, -1.295118, -2.629707, -0.787565, 1.570796, 1.697874],accel_mss,speed_ms,0,blend_radius_m)
    movel([0.126768, -1.295285, -2.629608, -0.787496, 1.570796, 1.697564],accel_mss,speed_ms,0,blend_radius_m)
    movel([0.126509, -1.295638, -2.629401, -0.787351, 1.570796, 1.697305],accel_mss,speed_ms,0,blend_radius_m)
    movel([0.126305, -1.295952, -2.629216, -0.787222, 1.570796, 1.697101],accel_mss,speed_ms,0,blend_radius_m)
    movel([0.126018, -1.296162, -2.629092, -0.787135, 1.570796, 1.696815],accel_mss,speed_ms,0,blend_radius_m)
    movel([0.125705, -1.296433, -2.628932, -0.787024, 1.570796, 1.696501],accel_mss,speed_ms,0,blend_radius_m)
    movel([0.125159, -1.297034, -2.628577, -0.786778, 1.570796, 1.695956],accel_mss,speed_ms,0,blend_radius_m)
    movel([0.125190, -1.296739, -2.628751, -0.786898, 1.570796, 1.695986],accel_mss,speed_ms,0,blend_radius_m)
    movel([0.125220, -1.296186, -2.629077, -0.787125, 1.570796, 1.696016],accel_mss,speed_ms,0,blend_radius_m)
    movel([0.125143, -1.295901, -2.629246, -0.787243, 1.570796, 1.695940],accel_mss,speed_ms,0,blend_radius_m)
    movel([0.124950, -1.295802, -2.629304, -0.787283, 1.570796, 1.695747],accel_mss,speed_ms,0,blend_radius_m)
    movel([0.124630, -1.295855, -2.629273, -0.787261, 1.570796, 1.695427],accel_mss,speed_ms,0,blend_radius_m)
    movel([0.124057, -1.296046, -2.629160, -0.787183, 1.570796, 1.694854],accel_mss,speed_ms,0,blend_radius_m)
    movel([0.123746, -1.295996, -2.629189, -0.787203, 1.570796, 1.694542],accel_mss,speed_ms,0,blend_radius_m)
    movel([0.123747, -1.295609, -2.629418, -0.787363, 1.570796, 1.694543],accel_mss,speed_ms,0,blend_radius_m)
    movel([0.123613, -1.295366, -2.629560, -0.787462, 1.570796, 1.694410],accel_mss,speed_ms,0,blend_radius_m)
    movel([0.123150, -1.295168, -2.629677, -0.787544, 1.570796, 1.693946],accel_mss,speed_ms,0,blend_radius_m)
    movel([0.123672, -1.294806, -2.629890, -0.787693, 1.570796, 1.694469],accel_mss,speed_ms,0,blend_radius_m)
    movel([0.124196, -1.294443, -2.630103, -0.787843, 1.570796, 1.694992],accel_mss,speed_ms,0,blend_radius_m)
    movel([0.124474, -1.294827, -2.629877, -0.787684, 1.570796, 1.695270],accel_mss,speed_ms,0,blend_radius_m)
    movel([0.124862, -1.295182, -2.629669, -0.787538, 1.570796, 1.695659],accel_mss,speed_ms,0,blend_radius_m)
    movel([0.125351, -1.295307, -2.629595, -0.787487, 1.570796, 1.696148],accel_mss,speed_ms,0,blend_radius_m)
    movel([0.125916, -1.295194, -2.629662, -0.787533, 1.570796, 1.696713],accel_mss,speed_ms,0,blend_radius_m)
    movel([0.126523, -1.294860, -2.629858, -0.787671, 1.570796, 1.697320],accel_mss,speed_ms,0,blend_radius_m)
    movel([0.126930, -1.294519, -2.630058, -0.787811, 1.570796, 1.697726],accel_mss,speed_ms,0,blend_radius_m)
    movel([0.127231, -1.294156, -2.630271, -0.787961, 1.570796, 1.698027],accel_mss,speed_ms,0,blend_radius_m)
    movel([0.127430, -1.293762, -2.630503, -0.788124, 1.570796, 1.698227],accel_mss,speed_ms,0,blend_radius_m)
    movel([0.127541, -1.293320, -2.630762, -0.788307, 1.570796, 1.698338],accel_mss,speed_ms,0,blend_radius_m)
    movel([0.127562, -1.293022, -2.630936, -0.788430, 1.570796, 1.698359],accel_mss,speed_ms,0,blend_radius_m)
    movel([0.127420, -1.292662, -2.631147, -0.788580, 1.570796, 1.698216],accel_mss,speed_ms,0,blend_radius_m)
    movel([0.127207, -1.292493, -2.631246, -0.788650, 1.570796, 1.698004],accel_mss,speed_ms,0,blend_radius_m)
    movel([0.126764, -1.292319, -2.631347, -0.788722, 1.570796, 1.697560],accel_mss,speed_ms,0,blend_radius_m)
    movel([0.126263, -1.292360, -2.631324, -0.788705, 1.570796, 1.697060],accel_mss,speed_ms,0,blend_radius_m)
    movel([0.125714, -1.292616, -2.631174, -0.788599, 1.570796, 1.696510],accel_mss,speed_ms,0,blend_radius_m)
    speed_ms = 0.003
    movel([0.125714, -1.278714, -2.624568, -0.809107, 1.570796, 1.696510],accel_mss,speed_ms,0,blend_radius_m)
    speed_ms = 1.000
    movel([0.125714, -1.252259, -2.610972, -0.849158, 1.570796, 1.696510],accel_mss,speed_ms,0,blend_radius_m)
    movel([0.133504, -1.250299, -2.612053, -0.850037, 1.570796, 1.704301],accel_mss,speed_ms,0,blend_radius_m)
    movel([0.133504, -1.276780, -2.625675, -0.809934, 1.570796, 1.704301],accel_mss,speed_ms,0,blend_radius_m)
    speed_ms = 0.003
    movel([0.133504, -1.287176, -2.630651, -0.794562, 1.570796, 1.704301],accel_mss,speed_ms,0,blend_radius_m)
    speed_ms = 0.007
    movel([0.134027, -1.286061, -2.631296, -0.795032, 1.570796, 1.704823],accel_mss,speed_ms,0,blend_radius_m)
    movel([0.134594, -1.284880, -2.631978, -0.795531, 1.570796, 1.705391],accel_mss,speed_ms,0,blend_radius_m)
    movel([0.135270, -1.283489, -2.632779, -0.796121, 1.570796, 1.706066],accel_mss,speed_ms,0,blend_radius_m)
    movel([0.136116, -1.281738, -2.633783, -0.796867, 1.570796, 1.706912],accel_mss,speed_ms,0,blend_radius_m)
    movel([0.136618, -1.280641, -2.634411, -0.797337, 1.570796, 1.707415],accel_mss,speed_ms,0,blend_radius_m)
    movel([0.136933, -1.279892, -2.634838, -0.797658, 1.570796, 1.707729],accel_mss,speed_ms,0,blend_radius_m)
    movel([0.136793, -1.279648, -2.634978, -0.797763, 1.570796, 1.707589],accel_mss,speed_ms,0,blend_radius_m)
    movel([0.136471, -1.279687, -2.634956, -0.797747, 1.570796, 1.707267],accel_mss,speed_ms,0,blend_radius_m)
    movel([0.135922, -1.279812, -2.634884, -0.797693, 1.570796, 1.706718],accel_mss,speed_ms,0,blend_radius_m)
    movel([0.134913, -1.280094, -2.634723, -0.797572, 1.570796, 1.705709],accel_mss,speed_ms,0,blend_radius_m)
    movel([0.133552, -1.280474, -2.634507, -0.797409, 1.570796, 1.704348],accel_mss,speed_ms,0,blend_radius_m)
    movel([0.133163, -1.280512, -2.634485, -0.797392, 1.570796, 1.703959],accel_mss,speed_ms,0,blend_radius_m)
    movel([0.133239, -1.279945, -2.634808, -0.797635, 1.570796, 1.704035],accel_mss,speed_ms,0,blend_radius_m)
    movel([0.133883, -1.278640, -2.635552, -0.798197, 1.570796, 1.704679],accel_mss,speed_ms,0,blend_radius_m)
    movel([0.134493, -1.277389, -2.636262, -0.798738, 1.570796, 1.705290],accel_mss,speed_ms,0,blend_radius_m)
    movel([0.135185, -1.275965, -2.637069, -0.799355, 1.570796, 1.705981],accel_mss,speed_ms,0,blend_radius_m)
    movel([0.135883, -1.274540, -2.637873, -0.799976, 1.570796, 1.706679],accel_mss,speed_ms,0,blend_radius_m)
    movel([0.136516, -1.273290, -2.638576, -0.800522, 1.570796, 1.707313],accel_mss,speed_ms,0,blend_radius_m)
    movel([0.137066, -1.272226, -2.639174, -0.800989, 1.570796, 1.707862],accel_mss,speed_ms,0,blend_radius_m)
    movel([0.137461, -1.271810, -2.639407, -0.801172, 1.570796, 1.708257],accel_mss,speed_ms,0,blend_radius_m)
    movel([0.137870, -1.271626, -2.639510, -0.801253, 1.570796, 1.708666],accel_mss,speed_ms,0,blend_radius_m)
    movel([0.138572, -1.271381, -2.639647, -0.801361, 1.570796, 1.709368],accel_mss,speed_ms,0,blend_radius_m)
    movel([0.140061, -1.270920, -2.639905, -0.801564, 1.570796, 1.710857],accel_mss,speed_ms,0,blend_radius_m)
    movel([0.141304, -1.270549, -2.640113, -0.801727, 1.570796, 1.712100],accel_mss,speed_ms,0,blend_radius_m)
    movel([0.142088, -1.270338, -2.640230, -0.801820, 1.570796, 1.712884],accel_mss,speed_ms,0,blend_radius_m)
    movel([0.142614, -1.270221, -2.640296, -0.801872, 1.570796, 1.713410],accel_mss,speed_ms,0,blend_radius_m)
    movel([0.142766, -1.270404, -2.640193, -0.801791, 1.570796, 1.713562],accel_mss,speed_ms,0,blend_radius_m)
    movel([0.142429, -1.271016, -2.639852, -0.801521, 1.570796, 1.713226],accel_mss,speed_ms,0,blend_radius_m)
    movel([0.141892, -1.271915, -2.639348, -0.801126, 1.570796, 1.712688],accel_mss,speed_ms,0,blend_radius_m)
    movel([0.140997, -1.273330, -2.638554, -0.800505, 1.570796, 1.711794],accel_mss,speed_ms,0,blend_radius_m)
    movel([0.140062, -1.274814, -2.637718, -0.799856, 1.570796, 1.710858],accel_mss,speed_ms,0,blend_radius_m)
    movel([0.139543, -1.275686, -2.637226, -0.799477, 1.570796, 1.710339],accel_mss,speed_ms,0,blend_radius_m)
    movel([0.139241, -1.276249, -2.636908, -0.799232, 1.570796, 1.710037],accel_mss,speed_ms,0,blend_radius_m)
    movel([0.139361, -1.276496, -2.636768, -0.799125, 1.570796, 1.710158],accel_mss,speed_ms,0,blend_radius_m)
    movel([0.139639, -1.276473, -2.636781, -0.799135, 1.570796, 1.710435],accel_mss,speed_ms,0,blend_radius_m)
    movel([0.140108, -1.276373, -2.636838, -0.799178, 1.570796, 1.710904],accel_mss,speed_ms,0,blend_radius_m)
    movel([0.140935, -1.276149, -2.636965, -0.799276, 1.570796, 1.711731],accel_mss,speed_ms,0,blend_radius_m)
    movel([0.141601, -1.275973, -2.637064, -0.799352, 1.570796, 1.712397],accel_mss,speed_ms,0,blend_radius_m)
    movel([0.142119, -1.275857, -2.637130, -0.799402, 1.570796, 1.712915],accel_mss,speed_ms,0,blend_radius_m)
    movel([0.142511, -1.275786, -2.637170, -0.799433, 1.570796, 1.713307],accel_mss,speed_ms,0,blend_radius_m)
    movel([0.139443, -1.280014, -2.634769, -0.797606, 1.570796, 1.710239],accel_mss,speed_ms,0,blend_radius_m)
    movel([0.136516, -1.283764, -2.632621, -0.796004, 1.570796, 1.707313],accel_mss,speed_ms,0,blend_radius_m)
    movel([0.134149, -1.286736, -2.630906, -0.794747, 1.570796, 1.704946],accel_mss,speed_ms,0,blend_radius_m)
    movel([0.133914, -1.286997, -2.630755, -0.794637, 1.570796, 1.704710],accel_mss,speed_ms,0,blend_radius_m)
    movel([0.133557, -1.287232, -2.630619, -0.794539, 1.570796, 1.704353],accel_mss,speed_ms,0,blend_radius_m)
    speed_ms = 0.003
    movel([0.133504, -1.290698, -2.632293, -0.789397, 1.570796, 1.704301],accel_mss,speed_ms,0,blend_radius_m)
    speed_ms = 0.007
    movel([0.134027, -1.289586, -2.632940, -0.789863, 1.570796, 1.704823],accel_mss,speed_ms,0,blend_radius_m)
    movel([0.134594, -1.288408, -2.633624, -0.790357, 1.570796, 1.705391],accel_mss,speed_ms,0,blend_radius_m)
    movel([0.135270, -1.287019, -2.634427, -0.790942, 1.570796, 1.706066],accel_mss,speed_ms,0,blend_radius_m)
    movel([0.136116, -1.285272, -2.635435, -0.791682, 1.570796, 1.706912],accel_mss,speed_ms,0,blend_radius_m)
    movel([0.136618, -1.284177, -2.636065, -0.792147, 1.570796, 1.707415],accel_mss,speed_ms,0,blend_radius_m)
    movel([0.136933, -1.283431, -2.636493, -0.792466, 1.570796, 1.707729],accel_mss,speed_ms,0,blend_radius_m)
    movel([0.136793, -1.283186, -2.636633, -0.792570, 1.570796, 1.707589],accel_mss,speed_ms,0,blend_radius_m)
    movel([0.136471, -1.283225, -2.636610, -0.792553, 1.570796, 1.707267],accel_mss,speed_ms,0,blend_radius_m)
    movel([0.135922, -1.283350, -2.636539, -0.792500, 1.570796, 1.706718],accel_mss,speed_ms,0,blend_radius_m)
    movel([0.134913, -1.283631, -2.636378, -0.792380, 1.570796, 1.705709],accel_mss,speed_ms,0,blend_radius_m)
    movel([0.133552, -1.284011, -2.636160, -0.792218, 1.570796, 1.704348],accel_mss,speed_ms,0,blend_radius_m)
    movel([0.133163, -1.284049, -2.636138, -0.792202, 1.570796, 1.703959],accel_mss,speed_ms,0,blend_radius_m)
    movel([0.133239, -1.283483, -2.636463, -0.792443, 1.570796, 1.704035],accel_mss,speed_ms,0,blend_radius_m)
    movel([0.133883, -1.282181, -2.637208, -0.793000, 1.570796, 1.704679],accel_mss,speed_ms,0,blend_radius_m)
    movel([0.134493, -1.280933, -2.637921, -0.793536, 1.570796, 1.705290],accel_mss,speed_ms,0,blend_radius_m)
    movel([0.135185, -1.279511, -2.638730, -0.794148, 1.570796, 1.705981],accel_mss,speed_ms,0,blend_radius_m)
    movel([0.135883, -1.278090, -2.639536, -0.794763, 1.570796, 1.706679],accel_mss,speed_ms,0,blend_radius_m)
    movel([0.136516, -1.276842, -2.640242, -0.795305, 1.570796, 1.707313],accel_mss,speed_ms,0,blend_radius_m)
    movel([0.137066, -1.275780, -2.640842, -0.795768, 1.570796, 1.707862],accel_mss,speed_ms,0,blend_radius_m)
    movel([0.137461, -1.275364, -2.641076, -0.795949, 1.570796, 1.708257],accel_mss,speed_ms,0,blend_radius_m)
    movel([0.137870, -1.275181, -2.641179, -0.796029, 1.570796, 1.708666],accel_mss,speed_ms,0,blend_radius_m)
    movel([0.138572, -1.274937, -2.641316, -0.796136, 1.570796, 1.709368],accel_mss,speed_ms,0,blend_radius_m)
    movel([0.140061, -1.274476, -2.641575, -0.796337, 1.570796, 1.710857],accel_mss,speed_ms,0,blend_radius_m)
    movel([0.141304, -1.274106, -2.641783, -0.796500, 1.570796, 1.712100],accel_mss,speed_ms,0,blend_radius_m)
    movel([0.142088, -1.273896, -2.641901, -0.796592, 1.570796, 1.712884],accel_mss,speed_ms,0,blend_radius_m)
    movel([0.142614, -1.273779, -2.641967, -0.796643, 1.570796, 1.713410],accel_mss,speed_ms,0,blend_radius_m)
    movel([0.142766, -1.273962, -2.641864, -0.796563, 1.570796, 1.713562],accel_mss,speed_ms,0,blend_radius_m)
    movel([0.142429, -1.274572, -2.641521, -0.796295, 1.570796, 1.713226],accel_mss,speed_ms,0,blend_radius_m)
    movel([0.141892, -1.275469, -2.641017, -0.795903, 1.570796, 1.712688],accel_mss,speed_ms,0,blend_radius_m)
    movel([0.140997, -1.276882, -2.640220, -0.795287, 1.570796, 1.711794],accel_mss,speed_ms,0,blend_radius_m)
    movel([0.140062, -1.278363, -2.639382, -0.794644, 1.570796, 1.710858],accel_mss,speed_ms,0,blend_radius_m)
    movel([0.139543, -1.279233, -2.638888, -0.794268, 1.570796, 1.710339],accel_mss,speed_ms,0,blend_radius_m)
    movel([0.139241, -1.279795, -2.638569, -0.794026, 1.570796, 1.710037],accel_mss,speed_ms,0,blend_radius_m)
    movel([0.139361, -1.280041, -2.638429, -0.793919, 1.570796, 1.710158],accel_mss,speed_ms,0,blend_radius_m)
    movel([0.139639, -1.280019, -2.638441, -0.793929, 1.570796, 1.710435],accel_mss,speed_ms,0,blend_radius_m)
    movel([0.140108, -1.279919, -2.638498, -0.793972, 1.570796, 1.710904],accel_mss,speed_ms,0,blend_radius_m)
    movel([0.140935, -1.279695, -2.638626, -0.794069, 1.570796, 1.711731],accel_mss,speed_ms,0,blend_radius_m)
    movel([0.141601, -1.279519, -2.638725, -0.794144, 1.570796, 1.712397],accel_mss,speed_ms,0,blend_radius_m)
    movel([0.142119, -1.279403, -2.638791, -0.794194, 1.570796, 1.712915],accel_mss,speed_ms,0,blend_radius_m)
    movel([0.142511, -1.279332, -2.638832, -0.794225, 1.570796, 1.713307],accel_mss,speed_ms,0,blend_radius_m)
    movel([0.139443, -1.283552, -2.636423, -0.792414, 1.570796, 1.710239],accel_mss,speed_ms,0,blend_radius_m)
    movel([0.136516, -1.287294, -2.634269, -0.790826, 1.570796, 1.707313],accel_mss,speed_ms,0,blend_radius_m)
    movel([0.134149, -1.290260, -2.632549, -0.789581, 1.570796, 1.704946],accel_mss,speed_ms,0,blend_radius_m)
    movel([0.133914, -1.290520, -2.632397, -0.789472, 1.570796, 1.704710],accel_mss,speed_ms,0,blend_radius_m)
    movel([0.133557, -1.290754, -2.632261, -0.789374, 1.570796, 1.704353],accel_mss,speed_ms,0,blend_radius_m)
    speed_ms = 0.003
    movel([0.133504, -1.276780, -2.625675, -0.809934, 1.570796, 1.704301],accel_mss,speed_ms,0,blend_radius_m)
    speed_ms = 1.000
    movel([0.133504, -1.250299, -2.612053, -0.850037, 1.570796, 1.704301],accel_mss,speed_ms,0,blend_radius_m)
    movel([0.134600, -1.250152, -2.612134, -0.850103, 1.570796, 1.705396],accel_mss,speed_ms,0,blend_radius_m)
    movel([0.134600, -1.276635, -2.625758, -0.809996, 1.570796, 1.705396],accel_mss,speed_ms,0,blend_radius_m)
    speed_ms = 0.003
    movel([0.134600, -1.287031, -2.630735, -0.794623, 1.570796, 1.705396],accel_mss,speed_ms,0,blend_radius_m)
    speed_ms = 0.007
    movel([0.134785, -1.286680, -2.630938, -0.794771, 1.570796, 1.705582],accel_mss,speed_ms,0,blend_radius_m)
    movel([0.134992, -1.286772, -2.630885, -0.794732, 1.570796, 1.705789],accel_mss,speed_ms,0,blend_radius_m)
    movel([0.134805, -1.287044, -2.630727, -0.794617, 1.570796, 1.705602],accel_mss,speed_ms,0,blend_radius_m)
    speed_ms = 0.003
    movel([0.134600, -1.290554, -2.632377, -0.789458, 1.570796, 1.705396],accel_mss,speed_ms,0,blend_radius_m)
    speed_ms = 0.007
    movel([0.134785, -1.290204, -2.632581, -0.789604, 1.570796, 1.705582],accel_mss,speed_ms,0,blend_radius_m)
    movel([0.134992, -1.290295, -2.632528, -0.789566, 1.570796, 1.705789],accel_mss,speed_ms,0,blend_radius_m)
    movel([0.134805, -1.290567, -2.632370, -0.789452, 1.570796, 1.705602],accel_mss,speed_ms,0,blend_radius_m)
    speed_ms = 0.003
    movel([0.134600, -1.276635, -2.625758, -0.809996, 1.570796, 1.705396],accel_mss,speed_ms,0,blend_radius_m)
    speed_ms = 1.000
    movel([0.134600, -1.250152, -2.612134, -0.850103, 1.570796, 1.705396],accel_mss,speed_ms,0,blend_radius_m)
    movel([0.121826, -1.262324, -2.605349, -0.844716, 1.570796, 1.692622],accel_mss,speed_ms,0,blend_radius_m)
    movel([0.121826, -1.288645, -2.618813, -0.804932, 1.570796, 1.692622],accel_mss,speed_ms,0,blend_radius_m)
    speed_ms = 0.003
    movel([0.121826, -1.298967, -2.623729, -0.789693, 1.570796, 1.692622],accel_mss,speed_ms,0,blend_radius_m)
    speed_ms = 0.007
    movel([0.121317, -1.299452, -2.623441, -0.789496, 1.570796, 1.692114],accel_mss,speed_ms,0,blend_radius_m)
    movel([0.119704, -1.300013, -2.623107, -0.789270, 1.570796, 1.690500],accel_mss,speed_ms,0,blend_radius_m)
    movel([0.118907, -1.300275, -2.622950, -0.789164, 1.570796, 1.689704],accel_mss,speed_ms,0,blend_radius_m)
    movel([0.118218, -1.300489, -2.622823, -0.789077, 1.570796, 1.689014],accel_mss,speed_ms,0,blend_radius_m)
    movel([0.117635, -1.300656, -2.622723, -0.789010, 1.570796, 1.688431],accel_mss,speed_ms,0,blend_radius_m)
    movel([0.117680, -1.300296, -2.622938, -0.789155, 1.570796, 1.688476],accel_mss,speed_ms,0,blend_radius_m)
    movel([0.118005, -1.299994, -2.623118, -0.789277, 1.570796, 1.688801],accel_mss,speed_ms,0,blend_radius_m)
    movel([0.118443, -1.299668, -2.623312, -0.789409, 1.570796, 1.689239],accel_mss,speed_ms,0,blend_radius_m)
    movel([0.119078, -1.299316, -2.623522, -0.789551, 1.570796, 1.689874],accel_mss,speed_ms,0,blend_radius_m)
    movel([0.119872, -1.299016, -2.623700, -0.789673, 1.570796, 1.690668],accel_mss,speed_ms,0,blend_radius_m)
    movel([0.120636, -1.298823, -2.623815, -0.789751, 1.570796, 1.691433],accel_mss,speed_ms,0,blend_radius_m)
    movel([0.121168, -1.298807, -2.623825, -0.789758, 1.570796, 1.691964],accel_mss,speed_ms,0,blend_radius_m)
    movel([0.121826, -1.298967, -2.623729, -0.789693, 1.570796, 1.692622],accel_mss,speed_ms,0,blend_radius_m)
    speed_ms = 0.003
    movel([0.121826, -1.302464, -2.625351, -0.784574, 1.570796, 1.692622],accel_mss,speed_ms,0,blend_radius_m)
    speed_ms = 0.007
    movel([0.121317, -1.302948, -2.625062, -0.784379, 1.570796, 1.692114],accel_mss,speed_ms,0,blend_radius_m)
    movel([0.119704, -1.303507, -2.624727, -0.784155, 1.570796, 1.690500],accel_mss,speed_ms,0,blend_radius_m)
    movel([0.118907, -1.303769, -2.624570, -0.784050, 1.570796, 1.689704],accel_mss,speed_ms,0,blend_radius_m)
    movel([0.118218, -1.303982, -2.624443, -0.783965, 1.570796, 1.689014],accel_mss,speed_ms,0,blend_radius_m)
    movel([0.117635, -1.304148, -2.624343, -0.783898, 1.570796, 1.688431],accel_mss,speed_ms,0,blend_radius_m)
    movel([0.117680, -1.303789, -2.624558, -0.784042, 1.570796, 1.688476],accel_mss,speed_ms,0,blend_radius_m)
    movel([0.118005, -1.303488, -2.624738, -0.784163, 1.570796, 1.688801],accel_mss,speed_ms,0,blend_radius_m)
    movel([0.118443, -1.303163, -2.624933, -0.784293, 1.570796, 1.689239],accel_mss,speed_ms,0,blend_radius_m)
    movel([0.119078, -1.302812, -2.625143, -0.784434, 1.570796, 1.689874],accel_mss,speed_ms,0,blend_radius_m)
    movel([0.119872, -1.302513, -2.625322, -0.784554, 1.570796, 1.690668],accel_mss,speed_ms,0,blend_radius_m)
    movel([0.120636, -1.302320, -2.625437, -0.784632, 1.570796, 1.691433],accel_mss,speed_ms,0,blend_radius_m)
    movel([0.121168, -1.302304, -2.625447, -0.784638, 1.570796, 1.691964],accel_mss,speed_ms,0,blend_radius_m)
    movel([0.121826, -1.302464, -2.625351, -0.784574, 1.570796, 1.692622],accel_mss,speed_ms,0,blend_radius_m)
    speed_ms = 0.003
    movel([0.121826, -1.288645, -2.618813, -0.804932, 1.570796, 1.692622],accel_mss,speed_ms,0,blend_radius_m)
    speed_ms = 1.000
    movel([0.121826, -1.262324, -2.605349, -0.844716, 1.570796, 1.692622],accel_mss,speed_ms,0,blend_radius_m)
    movel([0.120026, -1.261669, -2.605719, -0.845001, 1.570796, 1.690822],accel_mss,speed_ms,0,blend_radius_m)
    movel([0.120026, -1.287998, -2.619191, -0.805199, 1.570796, 1.690822],accel_mss,speed_ms,0,blend_radius_m)
    speed_ms = 0.003
    movel([0.120026, -1.298325, -2.624111, -0.789953, 1.570796, 1.690822],accel_mss,speed_ms,0,blend_radius_m)
    speed_ms = 0.007
    movel([0.119728, -1.298558, -2.623973, -0.789859, 1.570796, 1.690524],accel_mss,speed_ms,0,blend_radius_m)
    movel([0.119540, -1.298405, -2.624063, -0.789921, 1.570796, 1.690336],accel_mss,speed_ms,0,blend_radius_m)
    movel([0.119639, -1.297161, -2.624801, -0.790427, 1.570796, 1.690435],accel_mss,speed_ms,0,blend_radius_m)
    movel([0.119800, -1.295899, -2.625547, -0.790943, 1.570796, 1.690596],accel_mss,speed_ms,0,blend_radius_m)
    movel([0.120032, -1.295652, -2.625693, -0.791044, 1.570796, 1.690828],accel_mss,speed_ms,0,blend_radius_m)
    movel([0.120190, -1.295966, -2.625508, -0.790915, 1.570796, 1.690987],accel_mss,speed_ms,0,blend_radius_m)
    movel([0.120151, -1.296357, -2.625277, -0.790755, 1.570796, 1.690947],accel_mss,speed_ms,0,blend_radius_m)
    movel([0.120117, -1.296690, -2.625080, -0.790619, 1.570796, 1.690913],accel_mss,speed_ms,0,blend_radius_m)
    movel([0.120092, -1.297052, -2.624865, -0.790471, 1.570796, 1.690888],accel_mss,speed_ms,0,blend_radius_m)
    movel([0.120080, -1.297394, -2.624663, -0.790332, 1.570796, 1.690876],accel_mss,speed_ms,0,blend_radius_m)
    movel([0.120083, -1.297648, -2.624512, -0.790228, 1.570796, 1.690879],accel_mss,speed_ms,0,blend_radius_m)
    movel([0.120085, -1.298064, -2.624266, -0.790059, 1.570796, 1.690881],accel_mss,speed_ms,0,blend_radius_m)
    movel([0.120026, -1.298325, -2.624111, -0.789953, 1.570796, 1.690822],accel_mss,speed_ms,0,blend_radius_m)
    speed_ms = 0.003
    movel([0.120026, -1.301823, -2.625734, -0.784832, 1.570796, 1.690822],accel_mss,speed_ms,0,blend_radius_m)
    speed_ms = 0.007
    movel([0.119728, -1.302055, -2.625595, -0.784738, 1.570796, 1.690524],accel_mss,speed_ms,0,blend_radius_m)
    movel([0.119540, -1.301903, -2.625686, -0.784800, 1.570796, 1.690336],accel_mss,speed_ms,0,blend_radius_m)
    movel([0.119639, -1.300661, -2.626426, -0.785301, 1.570796, 1.690435],accel_mss,speed_ms,0,blend_radius_m)
    movel([0.119800, -1.299402, -2.627175, -0.785812, 1.570796, 1.690596],accel_mss,speed_ms,0,blend_radius_m)
    movel([0.120032, -1.299156, -2.627321, -0.785912, 1.570796, 1.690828],accel_mss,speed_ms,0,blend_radius_m)
    movel([0.120190, -1.299469, -2.627135, -0.785785, 1.570796, 1.690987],accel_mss,speed_ms,0,blend_radius_m)
    movel([0.120151, -1.299860, -2.626903, -0.785626, 1.570796, 1.690947],accel_mss,speed_ms,0,blend_radius_m)
    movel([0.120117, -1.300191, -2.626706, -0.785492, 1.570796, 1.690913],accel_mss,speed_ms,0,blend_radius_m)
    movel([0.120092, -1.300553, -2.626491, -0.785345, 1.570796, 1.690888],accel_mss,speed_ms,0,blend_radius_m)
    movel([0.120080, -1.300894, -2.626288, -0.785207, 1.570796, 1.690876],accel_mss,speed_ms,0,blend_radius_m)
    movel([0.120083, -1.301148, -2.626137, -0.785105, 1.570796, 1.690879],accel_mss,speed_ms,0,blend_radius_m)
    movel([0.120085, -1.301562, -2.625890, -0.784937, 1.570796, 1.690881],accel_mss,speed_ms,0,blend_radius_m)
    movel([0.120026, -1.301823, -2.625734, -0.784832, 1.570796, 1.690822],accel_mss,speed_ms,0,blend_radius_m)
    speed_ms = 0.003
    movel([0.120026, -1.287998, -2.619191, -0.805199, 1.570796, 1.690822],accel_mss,speed_ms,0,blend_radius_m)
    speed_ms = 1.000
    movel([0.120026, -1.261669, -2.605719, -0.845001, 1.570796, 1.690822],accel_mss,speed_ms,0,blend_radius_m)
    movel([0.116168, -1.271002, -2.600404, -0.840983, 1.570796, 1.686965],accel_mss,speed_ms,0,blend_radius_m)
    movel([0.116168, -1.297202, -2.613753, -0.801434, 1.570796, 1.686965],accel_mss,speed_ms,0,blend_radius_m)
    speed_ms = 0.003
    movel([0.116168, -1.307470, -2.618626, -0.786293, 1.570796, 1.686965],accel_mss,speed_ms,0,blend_radius_m)
    speed_ms = 0.007
    movel([0.116264, -1.307655, -2.618514, -0.786220, 1.570796, 1.687061],accel_mss,speed_ms,0,blend_radius_m)
    movel([0.116014, -1.307868, -2.618385, -0.786135, 1.570796, 1.686811],accel_mss,speed_ms,0,blend_radius_m)
    movel([0.115957, -1.307586, -2.618556, -0.786247, 1.570796, 1.686754],accel_mss,speed_ms,0,blend_radius_m)
    speed_ms = 0.003
    movel([0.116168, -1.310947, -2.620234, -0.781208, 1.570796, 1.686965],accel_mss,speed_ms,0,blend_radius_m)
    speed_ms = 0.007
    movel([0.116264, -1.311132, -2.620122, -0.781135, 1.570796, 1.687061],accel_mss,speed_ms,0,blend_radius_m)
    movel([0.116014, -1.311345, -2.619992, -0.781052, 1.570796, 1.686811],accel_mss,speed_ms,0,blend_radius_m)
    movel([0.115957, -1.311062, -2.620164, -0.781163, 1.570796, 1.686754],accel_mss,speed_ms,0,blend_radius_m)
    speed_ms = 0.003
    movel([0.116168, -1.297202, -2.613753, -0.801434, 1.570796, 1.686965],accel_mss,speed_ms,0,blend_radius_m)
    speed_ms = 1.000
    movel([0.116168, -1.271002, -2.600404, -0.840983, 1.570796, 1.686965],accel_mss,speed_ms,0,blend_radius_m)
    movel([0.116392, -1.270566, -2.600654, -0.841169, 1.570796, 1.687188],accel_mss,speed_ms,0,blend_radius_m)
    movel([0.116392, -1.296772, -2.614010, -0.801607, 1.570796, 1.687188],accel_mss,speed_ms,0,blend_radius_m)
    speed_ms = 0.003
    movel([0.116392, -1.307043, -2.618885, -0.786461, 1.570796, 1.687188],accel_mss,speed_ms,0,blend_radius_m)
    speed_ms = 0.007
    movel([0.116629, -1.307111, -2.618844, -0.786434, 1.570796, 1.687425],accel_mss,speed_ms,0,blend_radius_m)
    movel([0.116775, -1.307253, -2.618758, -0.786378, 1.570796, 1.687571],accel_mss,speed_ms,0,blend_radius_m)
    movel([0.116737, -1.307677, -2.618501, -0.786211, 1.570796, 1.687534],accel_mss,speed_ms,0,blend_radius_m)
    movel([0.116307, -1.308129, -2.618227, -0.786033, 1.570796, 1.687103],accel_mss,speed_ms,0,blend_radius_m)
    movel([0.116026, -1.308258, -2.618149, -0.785982, 1.570796, 1.686822],accel_mss,speed_ms,0,blend_radius_m)
    movel([0.115755, -1.308292, -2.618128, -0.785969, 1.570796, 1.686552],accel_mss,speed_ms,0,blend_radius_m)
    movel([0.115521, -1.308226, -2.618168, -0.785995, 1.570796, 1.686317],accel_mss,speed_ms,0,blend_radius_m)
    movel([0.115371, -1.308092, -2.618249, -0.786047, 1.570796, 1.686167],accel_mss,speed_ms,0,blend_radius_m)
    movel([0.115411, -1.307703, -2.618485, -0.786201, 1.570796, 1.686208],accel_mss,speed_ms,0,blend_radius_m)
    movel([0.115602, -1.307442, -2.618643, -0.786303, 1.570796, 1.686398],accel_mss,speed_ms,0,blend_radius_m)
    movel([0.115851, -1.307220, -2.618778, -0.786391, 1.570796, 1.686647],accel_mss,speed_ms,0,blend_radius_m)
    movel([0.116392, -1.307043, -2.618885, -0.786461, 1.570796, 1.687188],accel_mss,speed_ms,0,blend_radius_m)
    speed_ms = 0.003
    movel([0.116392, -1.310521, -2.620493, -0.781374, 1.570796, 1.687188],accel_mss,speed_ms,0,blend_radius_m)
    speed_ms = 0.007
    movel([0.116629, -1.310589, -2.620452, -0.781348, 1.570796, 1.687425],accel_mss,speed_ms,0,blend_radius_m)
    movel([0.116775, -1.310731, -2.620366, -0.781292, 1.570796, 1.687571],accel_mss,speed_ms,0,blend_radius_m)
    movel([0.116737, -1.311153, -2.620109, -0.781127, 1.570796, 1.687534],accel_mss,speed_ms,0,blend_radius_m)
    movel([0.116307, -1.311604, -2.619834, -0.780951, 1.570796, 1.687103],accel_mss,speed_ms,0,blend_radius_m)
    movel([0.116026, -1.311734, -2.619755, -0.780900, 1.570796, 1.686822],accel_mss,speed_ms,0,blend_radius_m)
    movel([0.115755, -1.311767, -2.619735, -0.780887, 1.570796, 1.686552],accel_mss,speed_ms,0,blend_radius_m)
    movel([0.115521, -1.311701, -2.619775, -0.780913, 1.570796, 1.686317],accel_mss,speed_ms,0,blend_radius_m)
    movel([0.115371, -1.311568, -2.619856, -0.780965, 1.570796, 1.686167],accel_mss,speed_ms,0,blend_radius_m)
    movel([0.115411, -1.311180, -2.620093, -0.781117, 1.570796, 1.686208],accel_mss,speed_ms,0,blend_radius_m)
    movel([0.115602, -1.310920, -2.620251, -0.781218, 1.570796, 1.686398],accel_mss,speed_ms,0,blend_radius_m)
    movel([0.115851, -1.310697, -2.620386, -0.781305, 1.570796, 1.686647],accel_mss,speed_ms,0,blend_radius_m)
    movel([0.116392, -1.310521, -2.620493, -0.781374, 1.570796, 1.687188],accel_mss,speed_ms,0,blend_radius_m)
    speed_ms = 0.003
    movel([0.116392, -1.296772, -2.614010, -0.801607, 1.570796, 1.687188],accel_mss,speed_ms,0,blend_radius_m)
    speed_ms = 1.000
    movel([0.116392, -1.270566, -2.600654, -0.841169, 1.570796, 1.687188],accel_mss,speed_ms,0,blend_radius_m)
    movel([0.116886, -1.270023, -2.600966, -0.841400, 1.570796, 1.687682],accel_mss,speed_ms,0,blend_radius_m)
    movel([0.116886, -1.296236, -2.614329, -0.801824, 1.570796, 1.687682],accel_mss,speed_ms,0,blend_radius_m)
    speed_ms = 0.003
    movel([0.116886, -1.306511, -2.619207, -0.786671, 1.570796, 1.687682],accel_mss,speed_ms,0,blend_radius_m)
    speed_ms = 0.007
    movel([0.117447, -1.307212, -2.618783, -0.786394, 1.570796, 1.688243],accel_mss,speed_ms,0,blend_radius_m)
    movel([0.117533, -1.307552, -2.618577, -0.786260, 1.570796, 1.688329],accel_mss,speed_ms,0,blend_radius_m)
    movel([0.117542, -1.307798, -2.618428, -0.786163, 1.570796, 1.688338],accel_mss,speed_ms,0,blend_radius_m)
    movel([0.117485, -1.308067, -2.618265, -0.786058, 1.570796, 1.688282],accel_mss,speed_ms,0,blend_radius_m)
    movel([0.117331, -1.308483, -2.618012, -0.785894, 1.570796, 1.688127],accel_mss,speed_ms,0,blend_radius_m)
    movel([0.116647, -1.309555, -2.617361, -0.785473, 1.570796, 1.687443],accel_mss,speed_ms,0,blend_radius_m)
    movel([0.115597, -1.310425, -2.616831, -0.785133, 1.570796, 1.686393],accel_mss,speed_ms,0,blend_radius_m)
    movel([0.114416, -1.310904, -2.616539, -0.784946, 1.570796, 1.685213],accel_mss,speed_ms,0,blend_radius_m)
    movel([0.113366, -1.310883, -2.616551, -0.784954, 1.570796, 1.684162],accel_mss,speed_ms,0,blend_radius_m)
    movel([0.112726, -1.310400, -2.616846, -0.785143, 1.570796, 1.683523],accel_mss,speed_ms,0,blend_radius_m)
    movel([0.112524, -1.309529, -2.617377, -0.785483, 1.570796, 1.683320],accel_mss,speed_ms,0,blend_radius_m)
    movel([0.112801, -1.308480, -2.618014, -0.785895, 1.570796, 1.683597],accel_mss,speed_ms,0,blend_radius_m)
    movel([0.113505, -1.307497, -2.618610, -0.786282, 1.570796, 1.684301],accel_mss,speed_ms,0,blend_radius_m)
    movel([0.114637, -1.306675, -2.619108, -0.786607, 1.570796, 1.685433],accel_mss,speed_ms,0,blend_radius_m)
    movel([0.115867, -1.306317, -2.619324, -0.786748, 1.570796, 1.686663],accel_mss,speed_ms,0,blend_radius_m)
    movel([0.116886, -1.306511, -2.619207, -0.786671, 1.570796, 1.687682],accel_mss,speed_ms,0,blend_radius_m)
    speed_ms = 0.003
    movel([0.116886, -1.309990, -2.620816, -0.781583, 1.570796, 1.687682],accel_mss,speed_ms,0,blend_radius_m)
    speed_ms = 0.007
    movel([0.117447, -1.310690, -2.620391, -0.781308, 1.570796, 1.688243],accel_mss,speed_ms,0,blend_radius_m)
    movel([0.117533, -1.311029, -2.620185, -0.781176, 1.570796, 1.688329],accel_mss,speed_ms,0,blend_radius_m)
    movel([0.117542, -1.311275, -2.620035, -0.781080, 1.570796, 1.688338],accel_mss,speed_ms,0,blend_radius_m)
    movel([0.117485, -1.311542, -2.619872, -0.780975, 1.570796, 1.688282],accel_mss,speed_ms,0,blend_radius_m)
    movel([0.117331, -1.311958, -2.619618, -0.780813, 1.570796, 1.688127],accel_mss,speed_ms,0,blend_radius_m)
    movel([0.116647, -1.313027, -2.618965, -0.780397, 1.570796, 1.687443],accel_mss,speed_ms,0,blend_radius_m)
    movel([0.115597, -1.313896, -2.618434, -0.780060, 1.570796, 1.686393],accel_mss,speed_ms,0,blend_radius_m)
    movel([0.114416, -1.314373, -2.618141, -0.779875, 1.570796, 1.685213],accel_mss,speed_ms,0,blend_radius_m)
    movel([0.113366, -1.314353, -2.618153, -0.779883, 1.570796, 1.684162],accel_mss,speed_ms,0,blend_radius_m)
    movel([0.112726, -1.313870, -2.618449, -0.780070, 1.570796, 1.683523],accel_mss,speed_ms,0,blend_radius_m)
    movel([0.112524, -1.313002, -2.618981, -0.780407, 1.570796, 1.683320],accel_mss,speed_ms,0,blend_radius_m)
    movel([0.112801, -1.311955, -2.619620, -0.780814, 1.570796, 1.683597],accel_mss,speed_ms,0,blend_radius_m)
    movel([0.113505, -1.310974, -2.620218, -0.781197, 1.570796, 1.684301],accel_mss,speed_ms,0,blend_radius_m)
    movel([0.114637, -1.310154, -2.620717, -0.781518, 1.570796, 1.685433],accel_mss,speed_ms,0,blend_radius_m)
    movel([0.115867, -1.309797, -2.620933, -0.781658, 1.570796, 1.686663],accel_mss,speed_ms,0,blend_radius_m)
    movel([0.116886, -1.309990, -2.620816, -0.781583, 1.570796, 1.687682],accel_mss,speed_ms,0,blend_radius_m)
    speed_ms = 0.003
    movel([0.116886, -1.296236, -2.614329, -0.801824, 1.570796, 1.687682],accel_mss,speed_ms,0,blend_radius_m)
    speed_ms = 1.000
    movel([0.116886, -1.270023, -2.600966, -0.841400, 1.570796, 1.687682],accel_mss,speed_ms,0,blend_radius_m)
    movel([0.117073, -1.269567, -2.601228, -0.841594, 1.570796, 1.687869],accel_mss,speed_ms,0,blend_radius_m)
    movel([0.117073, -1.295787, -2.614596, -0.802006, 1.570796, 1.687869],accel_mss,speed_ms,0,blend_radius_m)
    speed_ms = 0.003
    movel([0.117073, -1.306064, -2.619477, -0.786848, 1.570796, 1.687869],accel_mss,speed_ms,0,blend_radius_m)
    speed_ms = 0.007
    movel([0.117431, -1.306268, -2.619354, -0.786767, 1.570796, 1.688227],accel_mss,speed_ms,0,blend_radius_m)
    movel([0.117694, -1.306570, -2.619171, -0.786648, 1.570796, 1.688490],accel_mss,speed_ms,0,blend_radius_m)
    movel([0.117887, -1.306988, -2.618918, -0.786483, 1.570796, 1.688683],accel_mss,speed_ms,0,blend_radius_m)
    movel([0.117925, -1.307742, -2.618461, -0.786185, 1.570796, 1.688722],accel_mss,speed_ms,0,blend_radius_m)
    movel([0.117618, -1.308659, -2.617905, -0.785825, 1.570796, 1.688415],accel_mss,speed_ms,0,blend_radius_m)
    movel([0.117030, -1.309576, -2.617348, -0.785465, 1.570796, 1.687826],accel_mss,speed_ms,0,blend_radius_m)
    movel([0.116258, -1.310332, -2.616888, -0.785169, 1.570796, 1.687054],accel_mss,speed_ms,0,blend_radius_m)
    movel([0.114701, -1.311181, -2.616370, -0.784838, 1.570796, 1.685497],accel_mss,speed_ms,0,blend_radius_m)
    movel([0.113273, -1.311322, -2.616284, -0.784783, 1.570796, 1.684070],accel_mss,speed_ms,0,blend_radius_m)
    movel([0.112334, -1.310714, -2.616655, -0.785020, 1.570796, 1.683130],accel_mss,speed_ms,0,blend_radius_m)
    movel([0.112113, -1.309518, -2.617383, -0.785488, 1.570796, 1.682909],accel_mss,speed_ms,0,blend_radius_m)
    movel([0.112346, -1.308685, -2.617890, -0.785814, 1.570796, 1.683143],accel_mss,speed_ms,0,blend_radius_m)
    movel([0.112822, -1.307865, -2.618387, -0.786137, 1.570796, 1.683618],accel_mss,speed_ms,0,blend_radius_m)
    movel([0.113509, -1.307118, -2.618839, -0.786431, 1.570796, 1.684305],accel_mss,speed_ms,0,blend_radius_m)
    movel([0.114356, -1.306497, -2.619215, -0.786677, 1.570796, 1.685152],accel_mss,speed_ms,0,blend_radius_m)
    movel([0.114960, -1.306182, -2.619406, -0.786802, 1.570796, 1.685756],accel_mss,speed_ms,0,blend_radius_m)
    movel([0.115511, -1.305990, -2.619522, -0.786878, 1.570796, 1.686308],accel_mss,speed_ms,0,blend_radius_m)
    movel([0.116048, -1.305915, -2.619567, -0.786908, 1.570796, 1.686844],accel_mss,speed_ms,0,blend_radius_m)
    movel([0.116602, -1.305944, -2.619549, -0.786896, 1.570796, 1.687398],accel_mss,speed_ms,0,blend_radius_m)
    movel([0.117073, -1.306064, -2.619477, -0.786848, 1.570796, 1.687869],accel_mss,speed_ms,0,blend_radius_m)
    speed_ms = 0.003
    movel([0.117073, -1.309545, -2.621087, -0.781758, 1.570796, 1.687869],accel_mss,speed_ms,0,blend_radius_m)
    speed_ms = 0.007
    movel([0.117431, -1.309748, -2.620963, -0.781678, 1.570796, 1.688227],accel_mss,speed_ms,0,blend_radius_m)
    movel([0.117694, -1.310050, -2.620780, -0.781559, 1.570796, 1.688490],accel_mss,speed_ms,0,blend_radius_m)
    movel([0.117887, -1.310466, -2.620527, -0.781396, 1.570796, 1.688683],accel_mss,speed_ms,0,blend_radius_m)
    movel([0.117925, -1.311219, -2.620069, -0.781101, 1.570796, 1.688722],accel_mss,speed_ms,0,blend_radius_m)
    movel([0.117618, -1.312134, -2.619511, -0.780744, 1.570796, 1.688415],accel_mss,speed_ms,0,blend_radius_m)
    movel([0.117030, -1.313048, -2.618952, -0.780389, 1.570796, 1.687826],accel_mss,speed_ms,0,blend_radius_m)
    movel([0.116258, -1.313802, -2.618491, -0.780096, 1.570796, 1.687054],accel_mss,speed_ms,0,blend_radius_m)
    movel([0.114701, -1.314650, -2.617971, -0.779768, 1.570796, 1.685497],accel_mss,speed_ms,0,blend_radius_m)
    movel([0.113273, -1.314790, -2.617885, -0.779714, 1.570796, 1.684070],accel_mss,speed_ms,0,blend_radius_m)
    movel([0.112334, -1.314184, -2.618257, -0.779948, 1.570796, 1.683130],accel_mss,speed_ms,0,blend_radius_m)
    movel([0.112113, -1.312991, -2.618987, -0.780411, 1.570796, 1.682909],accel_mss,speed_ms,0,blend_radius_m)
    movel([0.112346, -1.312159, -2.619495, -0.780734, 1.570796, 1.683143],accel_mss,speed_ms,0,blend_radius_m)
    movel([0.112822, -1.311341, -2.619994, -0.781054, 1.570796, 1.683618],accel_mss,speed_ms,0,blend_radius_m)
    movel([0.113509, -1.310596, -2.620448, -0.781345, 1.570796, 1.684305],accel_mss,speed_ms,0,blend_radius_m)
    movel([0.114356, -1.309977, -2.620824, -0.781588, 1.570796, 1.685152],accel_mss,speed_ms,0,blend_radius_m)
    movel([0.114960, -1.309662, -2.621016, -0.781712, 1.570796, 1.685756],accel_mss,speed_ms,0,blend_radius_m)
    movel([0.115511, -1.309470, -2.621132, -0.781787, 1.570796, 1.686308],accel_mss,speed_ms,0,blend_radius_m)
    movel([0.116048, -1.309395, -2.621177, -0.781816, 1.570796, 1.686844],accel_mss,speed_ms,0,blend_radius_m)
    movel([0.116602, -1.309425, -2.621160, -0.781805, 1.570796, 1.687398],accel_mss,speed_ms,0,blend_radius_m)
    movel([0.117073, -1.309545, -2.621087, -0.781758, 1.570796, 1.687869],accel_mss,speed_ms,0,blend_radius_m)
    speed_ms = 0.003
    movel([0.117073, -1.295787, -2.614596, -0.802006, 1.570796, 1.687869],accel_mss,speed_ms,0,blend_radius_m)
    speed_ms = 1.000
    movel([0.117073, -1.269567, -2.601228, -0.841594, 1.570796, 1.687869],accel_mss,speed_ms,0,blend_radius_m)
    movel([0.122749, -1.268906, -2.601607, -0.841877, 1.570796, 1.693545],accel_mss,speed_ms,0,blend_radius_m)
    movel([0.122749, -1.295135, -2.614984, -0.802270, 1.570796, 1.693545],accel_mss,speed_ms,0,blend_radius_m)
    speed_ms = 0.003
    movel([0.122749, -1.305417, -2.619867, -0.787105, 1.570796, 1.693545],accel_mss,speed_ms,0,blend_radius_m)
    speed_ms = 0.007
    movel([0.123016, -1.305168, -2.620017, -0.787204, 1.570796, 1.693812],accel_mss,speed_ms,0,blend_radius_m)
    movel([0.123110, -1.305355, -2.619904, -0.787129, 1.570796, 1.693906],accel_mss,speed_ms,0,blend_radius_m)
    movel([0.122858, -1.305568, -2.619776, -0.787045, 1.570796, 1.693655],accel_mss,speed_ms,0,blend_radius_m)
    speed_ms = 0.003
    movel([0.122749, -1.308899, -2.621479, -0.782012, 1.570796, 1.693545],accel_mss,speed_ms,0,blend_radius_m)
    speed_ms = 0.007
    movel([0.123016, -1.308651, -2.621629, -0.782110, 1.570796, 1.693812],accel_mss,speed_ms,0,blend_radius_m)
    movel([0.123110, -1.308837, -2.621516, -0.782036, 1.570796, 1.693906],accel_mss,speed_ms,0,blend_radius_m)
    movel([0.122858, -1.309050, -2.621387, -0.781952, 1.570796, 1.693655],accel_mss,speed_ms,0,blend_radius_m)
    speed_ms = 0.003
    movel([0.122749, -1.295135, -2.614984, -0.802270, 1.570796, 1.693545],accel_mss,speed_ms,0,blend_radius_m)
    speed_ms = 1.000
    movel([0.122749, -1.268906, -2.601607, -0.841877, 1.570796, 1.693545],accel_mss,speed_ms,0,blend_radius_m)
    movel([0.122399, -1.268722, -2.601712, -0.841955, 1.570796, 1.693196],accel_mss,speed_ms,0,blend_radius_m)
    movel([0.122399, -1.294954, -2.615092, -0.802344, 1.570796, 1.693196],accel_mss,speed_ms,0,blend_radius_m)
    speed_ms = 0.003
    movel([0.122399, -1.305236, -2.619976, -0.787177, 1.570796, 1.693196],accel_mss,speed_ms,0,blend_radius_m)
    speed_ms = 0.007
    movel([0.122652, -1.304957, -2.620144, -0.787288, 1.570796, 1.693449],accel_mss,speed_ms,0,blend_radius_m)
    movel([0.122924, -1.304794, -2.620243, -0.787353, 1.570796, 1.693720],accel_mss,speed_ms,0,blend_radius_m)
    movel([0.123195, -1.304761, -2.620262, -0.787365, 1.570796, 1.693991],accel_mss,speed_ms,0,blend_radius_m)
    movel([0.123448, -1.304858, -2.620204, -0.787327, 1.570796, 1.694245],accel_mss,speed_ms,0,blend_radius_m)
    movel([0.123619, -1.305023, -2.620105, -0.787262, 1.570796, 1.694415],accel_mss,speed_ms,0,blend_radius_m)
    movel([0.123541, -1.305415, -2.619868, -0.787106, 1.570796, 1.694337],accel_mss,speed_ms,0,blend_radius_m)
    movel([0.123274, -1.305720, -2.619685, -0.786985, 1.570796, 1.694070],accel_mss,speed_ms,0,blend_radius_m)
    movel([0.122788, -1.306043, -2.619489, -0.786857, 1.570796, 1.693584],accel_mss,speed_ms,0,blend_radius_m)
    movel([0.122358, -1.306048, -2.619487, -0.786855, 1.570796, 1.693155],accel_mss,speed_ms,0,blend_radius_m)
    movel([0.122204, -1.305725, -2.619681, -0.786983, 1.570796, 1.693000],accel_mss,speed_ms,0,blend_radius_m)
    movel([0.122399, -1.305236, -2.619976, -0.787177, 1.570796, 1.693196],accel_mss,speed_ms,0,blend_radius_m)
    speed_ms = 0.003
    movel([0.122399, -1.308718, -2.621588, -0.782083, 1.570796, 1.693196],accel_mss,speed_ms,0,blend_radius_m)
    speed_ms = 0.007
    movel([0.122652, -1.308440, -2.621756, -0.782193, 1.570796, 1.693449],accel_mss,speed_ms,0,blend_radius_m)
    movel([0.122924, -1.308277, -2.621855, -0.782257, 1.570796, 1.693720],accel_mss,speed_ms,0,blend_radius_m)
    movel([0.123195, -1.308245, -2.621875, -0.782270, 1.570796, 1.693991],accel_mss,speed_ms,0,blend_radius_m)
    movel([0.123448, -1.308342, -2.621816, -0.782232, 1.570796, 1.694245],accel_mss,speed_ms,0,blend_radius_m)
    movel([0.123619, -1.308505, -2.621717, -0.782167, 1.570796, 1.694415],accel_mss,speed_ms,0,blend_radius_m)
    movel([0.123541, -1.308897, -2.621479, -0.782012, 1.570796, 1.694337],accel_mss,speed_ms,0,blend_radius_m)
    movel([0.123274, -1.309201, -2.621295, -0.781893, 1.570796, 1.694070],accel_mss,speed_ms,0,blend_radius_m)
    movel([0.122788, -1.309523, -2.621100, -0.781766, 1.570796, 1.693584],accel_mss,speed_ms,0,blend_radius_m)
    movel([0.122358, -1.309528, -2.621097, -0.781764, 1.570796, 1.693155],accel_mss,speed_ms,0,blend_radius_m)
    movel([0.122204, -1.309206, -2.621292, -0.781891, 1.570796, 1.693000],accel_mss,speed_ms,0,blend_radius_m)
    movel([0.122399, -1.308718, -2.621588, -0.782083, 1.570796, 1.693196],accel_mss,speed_ms,0,blend_radius_m)
    speed_ms = 0.003
    movel([0.122399, -1.294954, -2.615092, -0.802344, 1.570796, 1.693196],accel_mss,speed_ms,0,blend_radius_m)
    speed_ms = 1.000
    movel([0.122399, -1.268722, -2.601712, -0.841955, 1.570796, 1.693196],accel_mss,speed_ms,0,blend_radius_m)
    movel([0.122299, -1.268148, -2.602040, -0.842201, 1.570796, 1.693095],accel_mss,speed_ms,0,blend_radius_m)
    movel([0.122299, -1.294388, -2.615427, -0.802573, 1.570796, 1.693095],accel_mss,speed_ms,0,blend_radius_m)
    speed_ms = 0.003
    movel([0.122299, -1.304675, -2.620314, -0.787400, 1.570796, 1.693095],accel_mss,speed_ms,0,blend_radius_m)
    speed_ms = 0.007
    movel([0.123492, -1.303784, -2.620850, -0.787755, 1.570796, 1.694289],accel_mss,speed_ms,0,blend_radius_m)
    movel([0.124884, -1.303405, -2.621078, -0.787906, 1.570796, 1.695680],accel_mss,speed_ms,0,blend_radius_m)
    movel([0.125943, -1.303780, -2.620852, -0.787756, 1.570796, 1.696740],accel_mss,speed_ms,0,blend_radius_m)
    movel([0.126327, -1.304786, -2.620247, -0.787356, 1.570796, 1.697123],accel_mss,speed_ms,0,blend_radius_m)
    movel([0.125902, -1.306088, -2.619462, -0.786839, 1.570796, 1.696698],accel_mss,speed_ms,0,blend_radius_m)
    movel([0.125601, -1.306535, -2.619192, -0.786662, 1.570796, 1.696398],accel_mss,speed_ms,0,blend_radius_m)
    movel([0.125298, -1.306889, -2.618978, -0.786522, 1.570796, 1.696095],accel_mss,speed_ms,0,blend_radius_m)
    movel([0.124939, -1.307203, -2.618788, -0.786398, 1.570796, 1.695735],accel_mss,speed_ms,0,blend_radius_m)
    movel([0.124479, -1.307524, -2.618594, -0.786271, 1.570796, 1.695275],accel_mss,speed_ms,0,blend_radius_m)
    movel([0.123696, -1.307924, -2.618351, -0.786113, 1.570796, 1.694492],accel_mss,speed_ms,0,blend_radius_m)
    movel([0.122962, -1.308104, -2.618242, -0.786043, 1.570796, 1.693758],accel_mss,speed_ms,0,blend_radius_m)
    movel([0.122312, -1.308051, -2.618275, -0.786064, 1.570796, 1.693109],accel_mss,speed_ms,0,blend_radius_m)
    movel([0.121777, -1.307771, -2.618444, -0.786174, 1.570796, 1.692573],accel_mss,speed_ms,0,blend_radius_m)
    movel([0.121328, -1.306933, -2.618951, -0.786504, 1.570796, 1.692124],accel_mss,speed_ms,0,blend_radius_m)
    movel([0.121515, -1.305815, -2.619627, -0.786947, 1.570796, 1.692311],accel_mss,speed_ms,0,blend_radius_m)
    movel([0.122299, -1.304675, -2.620314, -0.787400, 1.570796, 1.693095],accel_mss,speed_ms,0,blend_radius_m)
    speed_ms = 0.003
    movel([0.122299, -1.308158, -2.621927, -0.782304, 1.570796, 1.693095],accel_mss,speed_ms,0,blend_radius_m)
    speed_ms = 0.007
    movel([0.123492, -1.307270, -2.622464, -0.782655, 1.570796, 1.694289],accel_mss,speed_ms,0,blend_radius_m)
    movel([0.124884, -1.306892, -2.622692, -0.782805, 1.570796, 1.695680],accel_mss,speed_ms,0,blend_radius_m)
    movel([0.125943, -1.307266, -2.622466, -0.782657, 1.570796, 1.696740],accel_mss,speed_ms,0,blend_radius_m)
    movel([0.126327, -1.308269, -2.621860, -0.782260, 1.570796, 1.697123],accel_mss,speed_ms,0,blend_radius_m)
    movel([0.125902, -1.309569, -2.621072, -0.781748, 1.570796, 1.696698],accel_mss,speed_ms,0,blend_radius_m)
    movel([0.125601, -1.310014, -2.620802, -0.781573, 1.570796, 1.696398],accel_mss,speed_ms,0,blend_radius_m)
    movel([0.125298, -1.310367, -2.620587, -0.781435, 1.570796, 1.696095],accel_mss,speed_ms,0,blend_radius_m)
    movel([0.124939, -1.310681, -2.620396, -0.781312, 1.570796, 1.695735],accel_mss,speed_ms,0,blend_radius_m)
    movel([0.124479, -1.311001, -2.620202, -0.781187, 1.570796, 1.695275],accel_mss,speed_ms,0,blend_radius_m)
    movel([0.123696, -1.311401, -2.619958, -0.781030, 1.570796, 1.694492],accel_mss,speed_ms,0,blend_radius_m)
    movel([0.122962, -1.311579, -2.619849, -0.780961, 1.570796, 1.693758],accel_mss,speed_ms,0,blend_radius_m)
    movel([0.122312, -1.311526, -2.619881, -0.780981, 1.570796, 1.693109],accel_mss,speed_ms,0,blend_radius_m)
    movel([0.121777, -1.311247, -2.620052, -0.781090, 1.570796, 1.692573],accel_mss,speed_ms,0,blend_radius_m)
    movel([0.121328, -1.310412, -2.620560, -0.781417, 1.570796, 1.692124],accel_mss,speed_ms,0,blend_radius_m)
    movel([0.121515, -1.309296, -2.621237, -0.781855, 1.570796, 1.692311],accel_mss,speed_ms,0,blend_radius_m)
    movel([0.122299, -1.308158, -2.621927, -0.782304, 1.570796, 1.693095],accel_mss,speed_ms,0,blend_radius_m)
    speed_ms = 0.003
    movel([0.122299, -1.294388, -2.615427, -0.802573, 1.570796, 1.693095],accel_mss,speed_ms,0,blend_radius_m)
    speed_ms = 1.000
    movel([0.122299, -1.268148, -2.602040, -0.842201, 1.570796, 1.693095],accel_mss,speed_ms,0,blend_radius_m)
    movel([0.122125, -1.267925, -2.602168, -0.842296, 1.570796, 1.692921],accel_mss,speed_ms,0,blend_radius_m)
    movel([0.122125, -1.294168, -2.615558, -0.802663, 1.570796, 1.692921],accel_mss,speed_ms,0,blend_radius_m)
    speed_ms = 0.003
    movel([0.122125, -1.304456, -2.620446, -0.787487, 1.570796, 1.692921],accel_mss,speed_ms,0,blend_radius_m)
    speed_ms = 0.007
    movel([0.122925, -1.303761, -2.620864, -0.787764, 1.570796, 1.693721],accel_mss,speed_ms,0,blend_radius_m)
    movel([0.123725, -1.303295, -2.621144, -0.787950, 1.570796, 1.694522],accel_mss,speed_ms,0,blend_radius_m)
    movel([0.124531, -1.303058, -2.621286, -0.788045, 1.570796, 1.695328],accel_mss,speed_ms,0,blend_radius_m)
    movel([0.125337, -1.303049, -2.621291, -0.788049, 1.570796, 1.696133],accel_mss,speed_ms,0,blend_radius_m)
    movel([0.125825, -1.303152, -2.621230, -0.788008, 1.570796, 1.696622],accel_mss,speed_ms,0,blend_radius_m)
    movel([0.126187, -1.303319, -2.621130, -0.787941, 1.570796, 1.696983],accel_mss,speed_ms,0,blend_radius_m)
    movel([0.126450, -1.303564, -2.620982, -0.787843, 1.570796, 1.697247],accel_mss,speed_ms,0,blend_radius_m)
    movel([0.126642, -1.303905, -2.620777, -0.787707, 1.570796, 1.697439],accel_mss,speed_ms,0,blend_radius_m)
    movel([0.126720, -1.304353, -2.620508, -0.787528, 1.570796, 1.697516],accel_mss,speed_ms,0,blend_radius_m)
    movel([0.126726, -1.304642, -2.620334, -0.787413, 1.570796, 1.697522],accel_mss,speed_ms,0,blend_radius_m)
    movel([0.126703, -1.304915, -2.620169, -0.787304, 1.570796, 1.697499],accel_mss,speed_ms,0,blend_radius_m)
    movel([0.126188, -1.306244, -2.619368, -0.786777, 1.570796, 1.696984],accel_mss,speed_ms,0,blend_radius_m)
    movel([0.125095, -1.307462, -2.618631, -0.786296, 1.570796, 1.695892],accel_mss,speed_ms,0,blend_radius_m)
    movel([0.123703, -1.308267, -2.618143, -0.785979, 1.570796, 1.694499],accel_mss,speed_ms,0,blend_radius_m)
    movel([0.122352, -1.308465, -2.618023, -0.785901, 1.570796, 1.693148],accel_mss,speed_ms,0,blend_radius_m)
    movel([0.121300, -1.308016, -2.618296, -0.786077, 1.570796, 1.692096],accel_mss,speed_ms,0,blend_radius_m)
    movel([0.120873, -1.307051, -2.618880, -0.786458, 1.570796, 1.691669],accel_mss,speed_ms,0,blend_radius_m)
    movel([0.121170, -1.305774, -2.619652, -0.786963, 1.570796, 1.691966],accel_mss,speed_ms,0,blend_radius_m)
    movel([0.122125, -1.304456, -2.620446, -0.787487, 1.570796, 1.692921],accel_mss,speed_ms,0,blend_radius_m)
    speed_ms = 0.003
    movel([0.122125, -1.307940, -2.622059, -0.782390, 1.570796, 1.692921],accel_mss,speed_ms,0,blend_radius_m)
    speed_ms = 0.007
    movel([0.122925, -1.307246, -2.622478, -0.782665, 1.570796, 1.693721],accel_mss,speed_ms,0,blend_radius_m)
    movel([0.123725, -1.306782, -2.622759, -0.782849, 1.570796, 1.694522],accel_mss,speed_ms,0,blend_radius_m)
    movel([0.124531, -1.306545, -2.622901, -0.782943, 1.570796, 1.695328],accel_mss,speed_ms,0,blend_radius_m)
    movel([0.125337, -1.306536, -2.622906, -0.782946, 1.570796, 1.696133],accel_mss,speed_ms,0,blend_radius_m)
    movel([0.125825, -1.306639, -2.622845, -0.782905, 1.570796, 1.696622],accel_mss,speed_ms,0,blend_radius_m)
    movel([0.126187, -1.306805, -2.622744, -0.782839, 1.570796, 1.696983],accel_mss,speed_ms,0,blend_radius_m)
    movel([0.126450, -1.307050, -2.622597, -0.782742, 1.570796, 1.697247],accel_mss,speed_ms,0,blend_radius_m)
    movel([0.126642, -1.307390, -2.622391, -0.782608, 1.570796, 1.697439],accel_mss,speed_ms,0,blend_radius_m)
    movel([0.126720, -1.307837, -2.622121, -0.782431, 1.570796, 1.697516],accel_mss,speed_ms,0,blend_radius_m)
    movel([0.126726, -1.308125, -2.621947, -0.782317, 1.570796, 1.697522],accel_mss,speed_ms,0,blend_radius_m)
    movel([0.126703, -1.308398, -2.621782, -0.782209, 1.570796, 1.697499],accel_mss,speed_ms,0,blend_radius_m)
    movel([0.126188, -1.309724, -2.620978, -0.781687, 1.570796, 1.696984],accel_mss,speed_ms,0,blend_radius_m)
    movel([0.125095, -1.310939, -2.620239, -0.781211, 1.570796, 1.695892],accel_mss,speed_ms,0,blend_radius_m)
    movel([0.123703, -1.311742, -2.619750, -0.780897, 1.570796, 1.694499],accel_mss,speed_ms,0,blend_radius_m)
    movel([0.122352, -1.311940, -2.619629, -0.780820, 1.570796, 1.693148],accel_mss,speed_ms,0,blend_radius_m)
    movel([0.121300, -1.311492, -2.619902, -0.780995, 1.570796, 1.692096],accel_mss,speed_ms,0,blend_radius_m)
    movel([0.120873, -1.310529, -2.620488, -0.781371, 1.570796, 1.691669],accel_mss,speed_ms,0,blend_radius_m)
    movel([0.121170, -1.309255, -2.621262, -0.781871, 1.570796, 1.691966],accel_mss,speed_ms,0,blend_radius_m)
    movel([0.122125, -1.307940, -2.622059, -0.782390, 1.570796, 1.692921],accel_mss,speed_ms,0,blend_radius_m)
    speed_ms = 0.003
    movel([0.122125, -1.294168, -2.615558, -0.802663, 1.570796, 1.692921],accel_mss,speed_ms,0,blend_radius_m)
    speed_ms = 1.000
    movel([0.122125, -1.267925, -2.602168, -0.842296, 1.570796, 1.692921],accel_mss,speed_ms,0,blend_radius_m)
    movel([0.121075, -1.274686, -2.598277, -0.839426, 1.570796, 1.691871],accel_mss,speed_ms,0,blend_radius_m)
    movel([0.121075, -1.300833, -2.611578, -0.799978, 1.570796, 1.691871],accel_mss,speed_ms,0,blend_radius_m)
    speed_ms = 0.003
    movel([0.121075, -1.311078, -2.616433, -0.784878, 1.570796, 1.691871],accel_mss,speed_ms,0,blend_radius_m)
    speed_ms = 0.007
    movel([0.123533, -1.310110, -2.617023, -0.785256, 1.570796, 1.694329],accel_mss,speed_ms,0,blend_radius_m)
    movel([0.125640, -1.309106, -2.617634, -0.785649, 1.570796, 1.696436],accel_mss,speed_ms,0,blend_radius_m)
    movel([0.127292, -1.308097, -2.618247, -0.786046, 1.570796, 1.698089],accel_mss,speed_ms,0,blend_radius_m)
    movel([0.127580, -1.307905, -2.618363, -0.786121, 1.570796, 1.698376],accel_mss,speed_ms,0,blend_radius_m)
    movel([0.127853, -1.307745, -2.618460, -0.786184, 1.570796, 1.698649],accel_mss,speed_ms,0,blend_radius_m)
    movel([0.128201, -1.307606, -2.618544, -0.786239, 1.570796, 1.698997],accel_mss,speed_ms,0,blend_radius_m)
    movel([0.128478, -1.307907, -2.618362, -0.786121, 1.570796, 1.699274],accel_mss,speed_ms,0,blend_radius_m)
    movel([0.128527, -1.308214, -2.618176, -0.786000, 1.570796, 1.699324],accel_mss,speed_ms,0,blend_radius_m)
    movel([0.128494, -1.308549, -2.617972, -0.785868, 1.570796, 1.699291],accel_mss,speed_ms,0,blend_radius_m)
    movel([0.128245, -1.308983, -2.617708, -0.785697, 1.570796, 1.699041],accel_mss,speed_ms,0,blend_radius_m)
    movel([0.127949, -1.309233, -2.617557, -0.785599, 1.570796, 1.698745],accel_mss,speed_ms,0,blend_radius_m)
    movel([0.127334, -1.309676, -2.617287, -0.785426, 1.570796, 1.698131],accel_mss,speed_ms,0,blend_radius_m)
    movel([0.126550, -1.310204, -2.616966, -0.785219, 1.570796, 1.697346],accel_mss,speed_ms,0,blend_radius_m)
    movel([0.126053, -1.310466, -2.616806, -0.785117, 1.570796, 1.696849],accel_mss,speed_ms,0,blend_radius_m)
    movel([0.125676, -1.310561, -2.616748, -0.785080, 1.570796, 1.696472],accel_mss,speed_ms,0,blend_radius_m)
    movel([0.125323, -1.310521, -2.616772, -0.785095, 1.570796, 1.696119],accel_mss,speed_ms,0,blend_radius_m)
    movel([0.125032, -1.310484, -2.616795, -0.785110, 1.570796, 1.695828],accel_mss,speed_ms,0,blend_radius_m)
    movel([0.124704, -1.310732, -2.616644, -0.785013, 1.570796, 1.695500],accel_mss,speed_ms,0,blend_radius_m)
    movel([0.124538, -1.311064, -2.616441, -0.784884, 1.570796, 1.695334],accel_mss,speed_ms,0,blend_radius_m)
    movel([0.124342, -1.311404, -2.616233, -0.784751, 1.570796, 1.695138],accel_mss,speed_ms,0,blend_radius_m)
    movel([0.123812, -1.311686, -2.616061, -0.784642, 1.570796, 1.694608],accel_mss,speed_ms,0,blend_radius_m)
    movel([0.123019, -1.311995, -2.615873, -0.784522, 1.570796, 1.693815],accel_mss,speed_ms,0,blend_radius_m)
    movel([0.122341, -1.312263, -2.615709, -0.784418, 1.570796, 1.693137],accel_mss,speed_ms,0,blend_radius_m)
    movel([0.121606, -1.312553, -2.615531, -0.784305, 1.570796, 1.692402],accel_mss,speed_ms,0,blend_radius_m)
    movel([0.119881, -1.313195, -2.615138, -0.784056, 1.570796, 1.690677],accel_mss,speed_ms,0,blend_radius_m)
    movel([0.118261, -1.313723, -2.614814, -0.783852, 1.570796, 1.689057],accel_mss,speed_ms,0,blend_radius_m)
    movel([0.116698, -1.314145, -2.614554, -0.783689, 1.570796, 1.687494],accel_mss,speed_ms,0,blend_radius_m)
    movel([0.115130, -1.314485, -2.614345, -0.783558, 1.570796, 1.685926],accel_mss,speed_ms,0,blend_radius_m)
